LIN {X 0,Y 574.65,Z 406.368,A -85,B 0,C 180,E1 -1993.417,E2 -1993.417} C_VEL
LIN {X 0,Y 574.045,Z 400.558,A -85,B 0,C 180,E1 -1993.505,E2 -1993.505} C_VEL
LIN {X 0,Y 573.916,Z 376.535,A -85,B 0,C 180,E1 -1993.811,E2 -1993.811} C_VEL
LIN {X 0,Y 573.362,Z 372.933,A -85,B 0,C 180,E1 -1993.874,E2 -1993.874} C_VEL
LIN {X 0,Y 573.52,Z 353.065,A -85,B 0,C 180,E1 -1996.97,E2 -1996.97} C_VEL
LIN {X 0,Y 573.745,Z 333.535,A -85,B 0,C 180,E1 -2000.059,E2 -2000.059} C_VEL
LIN {X 0,Y 573.574,Z 324.195,A -85,B 0,C 180,E1 -2001.567,E2 -2001.567} C_VEL
LIN {X 0,Y 573.285,Z 322.702,A -85,B 0,C 180,E1 -2001.838,E2 -2001.838} C_VEL
LIN {X 0,Y 573.272,Z 322.698,A -85,B 0,C 180,E1 -2004.878,E2 -2004.878} C_VEL
LIN {X 0,Y 573.27,Z 322.699,A -85,B 0,C 180,E1 -2007.766,E2 -2007.766} C_VEL
LIN {X 0,Y 573.249,Z 322.707,A -85,B 0,C 180,E1 -2010.176,E2 -2010.176} C_VEL
LIN {X 0,Y 573.257,Z 322.699,A -85,B 0,C 180,E1 -2012.645,E2 -2012.645} C_VEL
LIN {X 0,Y 573.209,Z 322.704,A -85,B 0,C 180,E1 -2015.188,E2 -2015.188} C_VEL
LIN {X 0,Y 573.234,Z 322.708,A -85,B 0,C 180,E1 -2017.808,E2 -2017.808} C_VEL
LIN {X 0,Y 573.25,Z 322.699,A -85,B 0,C 180,E1 -2020.525,E2 -2020.525} C_VEL
LIN {X 0,Y 573.24,Z 322.708,A -85,B 0,C 180,E1 -2023.668,E2 -2023.668} C_VEL
LIN {X 0,Y 573.212,Z 322.703,A -85,B 0,C 180,E1 -2026.638,E2 -2026.638} C_VEL
LIN {X 0,Y 573.25,Z 322.706,A -85,B 0,C 180,E1 -2029.475,E2 -2029.475} C_VEL
LIN {X 0,Y 573.22,Z 322.703,A -85,B 0,C 180,E1 -2032.19,E2 -2032.19} C_VEL
LIN {X 0,Y 573.227,Z 322.708,A -85,B 0,C 180,E1 -2035.23,E2 -2035.23} C_VEL
LIN {X 0,Y 573.223,Z 322.703,A -85,B 0,C 180,E1 -2038.183,E2 -2038.183} C_VEL
LIN {X 0,Y 573.229,Z 322.703,A -85,B 0,C 180,E1 -2040.631,E2 -2040.631} C_VEL
LIN {X 0,Y 573.188,Z 322.712,A -85,B 0,C 180,E1 -2043.518,E2 -2043.518} C_VEL
LIN {X 0,Y 573.189,Z 322.708,A -85,B 0,C 180,E1 -2046.132,E2 -2046.132} C_VEL
LIN {X 0,Y 573.225,Z 322.734,A -85,B 0,C 180,E1 -2047.471,E2 -2047.471} C_VEL
LIN {X 0,Y 573.941,Z 327.822,A -85,B 0,C 180,E1 -2048.258,E2 -2048.258} C_VEL
LIN {X 0,Y 573.725,Z 345.632,A -85,B 0,C 180,E1 -2050.871,E2 -2050.871} C_VEL
LIN {X 0,Y 573.558,Z 362.355,A -85,B 0,C 180,E1 -2053.29,E2 -2053.29} C_VEL
LIN {X 0,Y 574.612,Z 367.973,A -85,B 0,C 180,E1 -2053.394,E2 -2053.394} C_VEL
LIN {X 0,Y 574.27,Z 498.274,A -85,B 0,C 180,E1 -2055.062,E2 -2055.062} C_VEL
LIN {X 0,Y 574.177,Z 511.252,A -85,B 0,C 180,E1 -2055.339,E2 -2055.339} C_VEL
LIN {X 0,Y 574.09,Z 525.101,A -85,B 0,C 180,E1 -2055.771,E2 -2055.771} C_VEL
LIN {X 0,Y 573.918,Z 538.916,A -85,B 0,C 180,E1 -2056.365,E2 -2056.365} C_VEL
LIN {X 0,Y 573.741,Z 550.437,A -85,B 0,C 180,E1 -2056.991,E2 -2056.991} C_VEL
LIN {X 0,Y 573.601,Z 561.254,A -85,B 0,C 180,E1 -2057.708,E2 -2057.708} C_VEL
LIN {X 0,Y 573.455,Z 571.619,A -85,B 0,C 180,E1 -2058.53,E2 -2058.53} C_VEL
LIN {X 0,Y 573.355,Z 580.918,A -85,B 0,C 180,E1 -2059.404,E2 -2059.404} C_VEL
LIN {X 0,Y 573.256,Z 590.452,A -85,B 0,C 180,E1 -2060.472,E2 -2060.472} C_VEL
LIN {X 0,Y 573.143,Z 599.468,A -85,B 0,C 180,E1 -2061.715,E2 -2061.715} C_VEL
LIN {X 0,Y 573.091,Z 604.887,A -85,B 0,C 180,E1 -2062.601,E2 -2062.601} C_VEL
LIN {X 0,Y 573.022,Z 610.311,A -85,B 0,C 180,E1 -2063.662,E2 -2063.662} C_VEL
LIN {X 0,Y 573,Z 614.764,A -85,B 0,C 180,E1 -2064.721,E2 -2064.721} C_VEL
LIN {X 0,Y 573.029,Z 618.315,A -85,B 0,C 180,E1 -2065.779,E2 -2065.779} C_VEL
LIN {X 0,Y 572.957,Z 621.715,A -85,B 0,C 180,E1 -2067.187,E2 -2067.187} C_VEL
LIN {X 0,Y 572.939,Z 622.942,A -85,B 0,C 180,E1 -2067.89,E2 -2067.89} C_VEL
LIN {X 0,Y 572.936,Z 624.281,A -85,B 0,C 180,E1 -2069.296,E2 -2069.296} C_VEL
LIN {X 0,Y 572.937,Z 624.496,A -85,B 0,C 180,E1 -2069.999,E2 -2069.999} C_VEL
LIN {X 0,Y 572.941,Z 623.863,A -85,B 0,C 180,E1 -2071.405,E2 -2071.405} C_VEL
LIN {X 0,Y 572.954,Z 621.893,A -85,B 0,C 180,E1 -2072.811,E2 -2072.811} C_VEL
LIN {X 0,Y 573.008,Z 620.437,A -85,B 0,C 180,E1 -2073.515,E2 -2073.515} C_VEL
LIN {X 0,Y 572.955,Z 616.342,A -85,B 0,C 180,E1 -2074.925,E2 -2074.925} C_VEL
LIN {X 0,Y 573.044,Z 612.299,A -85,B 0,C 180,E1 -2075.983,E2 -2075.983} C_VEL
LIN {X 0,Y 573.052,Z 607.286,A -85,B 0,C 180,E1 -2077.043,E2 -2077.043} C_VEL
LIN {X 0,Y 573.128,Z 601.186,A -85,B 0,C 180,E1 -2078.106,E2 -2078.106} C_VEL
LIN {X 0,Y 573.219,Z 593.877,A -85,B 0,C 180,E1 -2079.17,E2 -2079.17} C_VEL
LIN {X 0,Y 573.303,Z 585.125,A -85,B 0,C 180,E1 -2080.238,E2 -2080.238} C_VEL
LIN {X 0,Y 573.486,Z 573.884,A -85,B 0,C 180,E1 -2081.365,E2 -2081.365} C_VEL
LIN {X 0,Y 573.584,Z 562.523,A -85,B 0,C 180,E1 -2082.291,E2 -2082.291} C_VEL
LIN {X 0,Y 573.731,Z 551.933,A -85,B 0,C 180,E1 -2083.007,E2 -2083.007} C_VEL
LIN {X 0,Y 573.879,Z 540.703,A -85,B 0,C 180,E1 -2083.634,E2 -2083.634} C_VEL
LIN {X 0,Y 574.011,Z 528.847,A -85,B 0,C 180,E1 -2084.173,E2 -2084.173} C_VEL
LIN {X 0,Y 574.173,Z 513.454,A -85,B 0,C 180,E1 -2084.696,E2 -2084.696} C_VEL
LIN {X 0,Y 574.271,Z 499.72,A -85,B 0,C 180,E1 -2085.004,E2 -2085.004} C_VEL
LIN {X 0,Y 574.432,Z 453.324,A -85,B 0,C 180,E1 -2085.613,E2 -2085.613} C_VEL
LIN {X 0,Y 574.556,Z 367.642,A -85,B 0,C 180,E1 -2086.702,E2 -2086.702} C_VEL
LIN {X 0,Y 573.565,Z 362.258,A -85,B 0,C 180,E1 -2086.813,E2 -2086.813} C_VEL
LIN {X 0,Y 573.811,Z 341.174,A -85,B 0,C 180,E1 -2089.868,E2 -2089.868} C_VEL
LIN {X 0,Y 573.911,Z 327.171,A -85,B 0,C 180,E1 -2091.93,E2 -2091.93} C_VEL
LIN {X 0,Y 573.224,Z 322.71,A -85,B 0,C 180,E1 -2092.646,E2 -2092.646} C_VEL
LIN {X 0,Y 573.215,Z 322.707,A -85,B 0,C 180,E1 -2095.41,E2 -2095.41} C_VEL
LIN {X 0,Y 573.193,Z 322.71,A -85,B 0,C 180,E1 -2098.565,E2 -2098.565} C_VEL
LIN {X 0,Y 573.205,Z 322.714,A -85,B 0,C 180,E1 -2100.993,E2 -2100.993} C_VEL
LIN {X 0,Y 573.235,Z 322.703,A -85,B 0,C 180,E1 -2103.519,E2 -2103.519} C_VEL
LIN {X 0,Y 573.184,Z 322.707,A -85,B 0,C 180,E1 -2106.052,E2 -2106.052} C_VEL
LIN {X 0,Y 573.222,Z 322.708,A -85,B 0,C 180,E1 -2108.701,E2 -2108.701} C_VEL
LIN {X 0,Y 573.192,Z 322.707,A -85,B 0,C 180,E1 -2111.458,E2 -2111.458} C_VEL
LIN {X 0,Y 573.206,Z 322.705,A -85,B 0,C 180,E1 -2114.334,E2 -2114.334} C_VEL
LIN {X 0,Y 573.218,Z 322.708,A -85,B 0,C 180,E1 -2116.639,E2 -2116.639} C_VEL
LIN {X 0,Y 573.234,Z 322.701,A -85,B 0,C 180,E1 -2119.474,E2 -2119.474} C_VEL
LIN {X 0,Y 573.209,Z 322.703,A -85,B 0,C 180,E1 -2122.19,E2 -2122.19} C_VEL
LIN {X 0,Y 573.208,Z 322.706,A -85,B 0,C 180,E1 -2125.23,E2 -2125.23} C_VEL
LIN {X 0,Y 573.223,Z 322.699,A -85,B 0,C 180,E1 -2127.773,E2 -2127.773} C_VEL
LIN {X 0,Y 573.218,Z 322.71,A -85,B 0,C 180,E1 -2130.631,E2 -2130.631} C_VEL
LIN {X 0,Y 573.194,Z 322.702,A -85,B 0,C 180,E1 -2133.513,E2 -2133.513} C_VEL
LIN {X 0,Y 573.181,Z 322.708,A -85,B 0,C 180,E1 -2136.132,E2 -2136.132} C_VEL
LIN {X 0,Y 573.236,Z 322.708,A -85,B 0,C 180,E1 -2138.709,E2 -2138.709} C_VEL
LIN {X 0,Y 573.183,Z 322.705,A -85,B 0,C 180,E1 -2141.41,E2 -2141.41} C_VEL
LIN {X 0,Y 573.206,Z 322.703,A -85,B 0,C 180,E1 -2143.62,E2 -2143.62} C_VEL
LIN {X 0,Y 573.182,Z 322.714,A -85,B 0,C 180,E1 -2146.528,E2 -2146.528} C_VEL
LIN {X 0,Y 573.22,Z 322.702,A -85,B 0,C 180,E1 -2149.402,E2 -2149.402} C_VEL
LIN {X 0,Y 573.244,Z 322.702,A -85,B 0,C 180,E1 -2152.249,E2 -2152.249} C_VEL
LIN {X 0,Y 573.266,Z 322.698,A -85,B 0,C 180,E1 -2155.077,E2 -2155.077} C_VEL
LIN {X 0,Y 573.27,Z 322.696,A -85,B 0,C 180,E1 -2157.892,E2 -2157.892} C_VEL
LIN {X 0,Y 573.316,Z 322.697,A -85,B 0,C 180,E1 -2160.702,E2 -2160.702} C_VEL
LIN {X 0,Y 573.282,Z 322.699,A -85,B 0,C 180,E1 -2162.811,E2 -2162.811} C_VEL
LIN {X 0,Y 573.243,Z 322.698,A -85,B 0,C 180,E1 -2165.629,E2 -2165.629} C_VEL
LIN {X 0,Y 573.22,Z 322.711,A -85,B 0,C 180,E1 -2168.46,E2 -2168.46} C_VEL
LIN {X 0,Y 573.219,Z 322.702,A -85,B 0,C 180,E1 -2171.313,E2 -2171.313} C_VEL
LIN {X 0,Y 573.261,Z 322.706,A -85,B 0,C 180,E1 -2174.423,E2 -2174.423} C_VEL
LIN {X 0,Y 573.202,Z 322.704,A -85,B 0,C 180,E1 -2177.113,E2 -2177.113} C_VEL
LIN {X 0,Y 573.219,Z 322.706,A -85,B 0,C 180,E1 -2180.078,E2 -2180.078} C_VEL
LIN {X 0,Y 573.21,Z 322.71,A -85,B 0,C 180,E1 -2182.339,E2 -2182.339} C_VEL
LIN {X 0,Y 573.193,Z 322.708,A -85,B 0,C 180,E1 -2184.866,E2 -2184.866} C_VEL
LIN {X 0,Y 573.216,Z 322.703,A -85,B 0,C 180,E1 -2187.769,E2 -2187.769} C_VEL
LIN {X 0,Y 573.209,Z 322.708,A -85,B 0,C 180,E1 -2190.178,E2 -2190.178} C_VEL
LIN {X 0,Y 573.231,Z 322.705,A -85,B 0,C 180,E1 -2192.647,E2 -2192.647} C_VEL
LIN {X 0,Y 573.169,Z 322.708,A -85,B 0,C 180,E1 -2195.191,E2 -2195.191} C_VEL
LIN {X 0,Y 573.202,Z 322.707,A -85,B 0,C 180,E1 -2197.81,E2 -2197.81} C_VEL
LIN {X 0,Y 573.188,Z 322.711,A -85,B 0,C 180,E1 -2200.53,E2 -2200.53} C_VEL
LIN {X 0,Y 573.186,Z 322.706,A -85,B 0,C 180,E1 -2203.364,E2 -2203.364} C_VEL
LIN {X 0,Y 573.182,Z 322.715,A -85,B 0,C 180,E1 -2206.338,E2 -2206.338} C_VEL
LIN {X 0,Y 573.178,Z 322.712,A -85,B 0,C 180,E1 -2208.54,E2 -2208.54} C_VEL
LIN {X 0,Y 573.204,Z 322.704,A -85,B 0,C 180,E1 -2211.297,E2 -2211.297} C_VEL
LIN {X 0,Y 573.173,Z 322.715,A -85,B 0,C 180,E1 -2214.024,E2 -2214.024} C_VEL
LIN {X 0,Y 573.213,Z 322.708,A -85,B 0,C 180,E1 -2216.516,E2 -2216.516} C_VEL
LIN {X 0,Y 573.209,Z 322.703,A -85,B 0,C 180,E1 -2219.121,E2 -2219.121} C_VEL
LIN {X 0,Y 573.184,Z 322.714,A -85,B 0,C 180,E1 -2221.984,E2 -2221.984} C_VEL
LIN {X 0,Y 573.199,Z 322.71,A -85,B 0,C 180,E1 -2224.589,E2 -2224.589} C_VEL
LIN {X 0,Y 573.241,Z 322.841,A -85,B 0,C 180,E1 -2226.382,E2 -2226.382} C_VEL
LIN {X 0,Y 574.048,Z 327.852,A -85,B 0,C 180,E1 -2227.127,E2 -2227.127} C_VEL
LIN {X 0,Y 573.904,Z 345.308,A -85,B 0,C 180,E1 -2229.575,E2 -2229.575} C_VEL
LIN {X 0,Y 573.681,Z 367.06,A -85,B 0,C 180,E1 -2232.572,E2 -2232.572} C_VEL
LIN {X 0,Y 573.602,Z 371.957,A -85,B 0,C 180,E1 -2233.239,E2 -2233.239} C_VEL
LIN {X 0,Y 574.57,Z 377.542,A -85,B 0,C 180,E1 -2233.342,E2 -2233.342} C_VEL
LIN {X 0,Y 574.302,Z 508.713,A -85,B 0,C 180,E1 -2235.019,E2 -2235.019} C_VEL
LIN {X 0,Y 574.171,Z 523.157,A -85,B 0,C 180,E1 -2235.341,E2 -2235.341} C_VEL
LIN {X 0,Y 574.023,Z 537.735,A -85,B 0,C 180,E1 -2235.827,E2 -2235.827} C_VEL
LIN {X 0,Y 573.874,Z 551.669,A -85,B 0,C 180,E1 -2236.456,E2 -2236.456} C_VEL
LIN {X 0,Y 573.718,Z 564.121,A -85,B 0,C 180,E1 -2237.173,E2 -2237.173} C_VEL
LIN {X 0,Y 573.532,Z 576.658,A -85,B 0,C 180,E1 -2238.067,E2 -2238.067} C_VEL
LIN {X 0,Y 573.435,Z 588.188,A -85,B 0,C 180,E1 -2239.085,E2 -2239.085} C_VEL
LIN {X 0,Y 573.239,Z 597.861,A -85,B 0,C 180,E1 -2240.118,E2 -2240.118} C_VEL
LIN {X 0,Y 573.201,Z 606.18,A -85,B 0,C 180,E1 -2241.185,E2 -2241.185} C_VEL
LIN {X 0,Y 573.109,Z 614.134,A -85,B 0,C 180,E1 -2242.426,E2 -2242.426} C_VEL
LIN {X 0,Y 573.02,Z 620.532,A -85,B 0,C 180,E1 -2243.664,E2 -2243.664} C_VEL
LIN {X 0,Y 573.001,Z 624.964,A -85,B 0,C 180,E1 -2244.723,E2 -2244.723} C_VEL
LIN {X 0,Y 573.028,Z 628.448,A -85,B 0,C 180,E1 -2245.781,E2 -2245.781} C_VEL
LIN {X 0,Y 572.956,Z 631.836,A -85,B 0,C 180,E1 -2247.189,E2 -2247.189} C_VEL
LIN {X 0,Y 572.941,Z 633.834,A -85,B 0,C 180,E1 -2248.595,E2 -2248.595} C_VEL
LIN {X 0,Y 572.937,Z 634.5,A -85,B 0,C 180,E1 -2250.001,E2 -2250.001} C_VEL
LIN {X 0,Y 572.941,Z 633.831,A -85,B 0,C 180,E1 -2251.407,E2 -2251.407} C_VEL
LIN {X 0,Y 572.956,Z 631.83,A -85,B 0,C 180,E1 -2252.813,E2 -2252.813} C_VEL
LIN {X 0,Y 573.028,Z 628.44,A -85,B 0,C 180,E1 -2254.221,E2 -2254.221} C_VEL
LIN {X 0,Y 573.055,Z 623.565,A -85,B 0,C 180,E1 -2255.631,E2 -2255.631} C_VEL
LIN {X 0,Y 573.059,Z 618.849,A -85,B 0,C 180,E1 -2256.694,E2 -2256.694} C_VEL
LIN {X 0,Y 573.126,Z 612.031,A -85,B 0,C 180,E1 -2257.93,E2 -2257.93} C_VEL
LIN {X 0,Y 573.226,Z 603.551,A -85,B 0,C 180,E1 -2259.172,E2 -2259.172} C_VEL
LIN {X 0,Y 573.305,Z 594.698,A -85,B 0,C 180,E1 -2260.24,E2 -2260.24} C_VEL
LIN {X 0,Y 573.464,Z 583.98,A -85,B 0,C 180,E1 -2261.309,E2 -2261.309} C_VEL
LIN {X 0,Y 573.618,Z 573.129,A -85,B 0,C 180,E1 -2262.202,E2 -2262.202} C_VEL
LIN {X 0,Y 573.74,Z 561.241,A -85,B 0,C 180,E1 -2263.009,E2 -2263.009} C_VEL
LIN {X 0,Y 573.957,Z 548.078,A -85,B 0,C 180,E1 -2263.725,E2 -2263.725} C_VEL
LIN {X 0,Y 574.104,Z 534.807,A -85,B 0,C 180,E1 -2264.285,E2 -2264.285} C_VEL
LIN {X 0,Y 574.204,Z 520.768,A -85,B 0,C 180,E1 -2264.721,E2 -2264.721} C_VEL
LIN {X 0,Y 574.309,Z 507.071,A -85,B 0,C 180,E1 -2265.005,E2 -2265.005} C_VEL
LIN {X 0,Y 574.472,Z 376.673,A -85,B 0,C 180,E1 -2266.672,E2 -2266.672} C_VEL
LIN {X 0,Y 573.592,Z 371.839,A -85,B 0,C 180,E1 -2266.777,E2 -2266.777} C_VEL
LIN {X 0,Y 573.841,Z 350.931,A -85,B 0,C 180,E1 -2269.646,E2 -2269.646} C_VEL
LIN {X 0,Y 574.092,Z 330.521,A -85,B 0,C 180,E1 -2272.493,E2 -2272.493} C_VEL
LIN {X 0,Y 573.715,Z 325.251,A -85,B 0,C 180,E1 -2273.256,E2 -2273.256} C_VEL
LIN {X 0,Y 573.228,Z 322.711,A -85,B 0,C 180,E1 -2273.643,E2 -2273.643} C_VEL
LIN {X 0,Y 573.201,Z 322.707,A -85,B 0,C 180,E1 -2276.485,E2 -2276.485} C_VEL
LIN {X 0,Y 573.225,Z 322.709,A -85,B 0,C 180,E1 -2279.369,E2 -2279.369} C_VEL
LIN {X 0,Y 573.241,Z 322.701,A -85,B 0,C 180,E1 -2282.226,E2 -2282.226} C_VEL
LIN {X 0,Y 573.234,Z 322.703,A -85,B 0,C 180,E1 -2284.771,E2 -2284.771} C_VEL
LIN {X 0,Y 573.234,Z 322.702,A -85,B 0,C 180,E1 -2287.808,E2 -2287.808} C_VEL
LIN {X 0,Y 573.249,Z 322.701,A -85,B 0,C 180,E1 -2290.526,E2 -2290.526} C_VEL
LIN {X 0,Y 573.241,Z 322.703,A -85,B 0,C 180,E1 -2293.36,E2 -2293.36} C_VEL
LIN {X 0,Y 573.249,Z 322.702,A -85,B 0,C 180,E1 -2296.331,E2 -2296.331} C_VEL
LIN {X 0,Y 573.234,Z 322.708,A -85,B 0,C 180,E1 -2298.543,E2 -2298.543} C_VEL
LIN {X 0,Y 573.242,Z 322.7,A -85,B 0,C 180,E1 -2301.298,E2 -2301.298} C_VEL
LIN {X 0,Y 573.198,Z 322.709,A -85,B 0,C 180,E1 -2304.021,E2 -2304.021} C_VEL
LIN {X 0,Y 573.274,Z 322.702,A -85,B 0,C 180,E1 -2306.518,E2 -2306.518} C_VEL
LIN {X 0,Y 573.23,Z 322.702,A -85,B 0,C 180,E1 -2309.119,E2 -2309.119} C_VEL
LIN {X 0,Y 573.227,Z 322.705,A -85,B 0,C 180,E1 -2311.435,E2 -2311.435} C_VEL
LIN {X 0,Y 573.225,Z 322.704,A -85,B 0,C 180,E1 -2314.589,E2 -2314.589} C_VEL
LIN {X 0,Y 573.221,Z 322.712,A -85,B 0,C 180,E1 -2317.662,E2 -2317.662} C_VEL
LIN {X 0,Y 573.233,Z 322.723,A -85,B 0,C 180,E1 -2318.278,E2 -2318.278} C_VEL
LIN {X 0,Y 573.78,Z 328.306,A -85,B 0,C 180,E1 -2319.194,E2 -2319.194} C_VEL
LIN {X 0,Y 573.558,Z 346.975,A -85,B 0,C 180,E1 -2322.162,E2 -2322.162} C_VEL
LIN {X 0,Y 573.397,Z 365.644,A -85,B 0,C 180,E1 -2325.085,E2 -2325.085} C_VEL
LIN {X 0,Y 573.36,Z 372.937,A -85,B 0,C 180,E1 -2326.216,E2 -2326.216} C_VEL
LIN {X 0,Y 574.089,Z 378.02,A -85,B 0,C 180,E1 -2326.302,E2 -2326.302} C_VEL
LIN {X 0,Y 573.881,Z 480.361,A -85,B 0,C 180,E1 -2327.602,E2 -2327.602} C_VEL
LIN {X 0,Y 573.814,Z 493.729,A -85,B 0,C 180,E1 -2327.915,E2 -2327.915} C_VEL
LIN {X 0,Y 573.704,Z 505.856,A -85,B 0,C 180,E1 -2328.339,E2 -2328.339} C_VEL
LIN {X 0,Y 573.62,Z 517.359,A -85,B 0,C 180,E1 -2328.878,E2 -2328.878} C_VEL
LIN {X 0,Y 573.437,Z 529.062,A -85,B 0,C 180,E1 -2329.585,E2 -2329.585} C_VEL
LIN {X 0,Y 573.329,Z 539.551,A -85,B 0,C 180,E1 -2330.386,E2 -2330.386} C_VEL
LIN {X 0,Y 573.243,Z 548.164,A -85,B 0,C 180,E1 -2331.185,E2 -2331.185} C_VEL
LIN {X 0,Y 573.162,Z 556.072,A -85,B 0,C 180,E1 -2332.071,E2 -2332.071} C_VEL
LIN {X 0,Y 573.089,Z 564.072,A -85,B 0,C 180,E1 -2333.169,E2 -2333.169} C_VEL
LIN {X 0,Y 573.071,Z 570.943,A -85,B 0,C 180,E1 -2334.37,E2 -2334.37} C_VEL
LIN {X 0,Y 573.028,Z 575.704,A -85,B 0,C 180,E1 -2335.428,E2 -2335.428} C_VEL
LIN {X 0,Y 573.023,Z 579.31,A -85,B 0,C 180,E1 -2336.484,E2 -2336.484} C_VEL
LIN {X 0,Y 572.959,Z 581.18,A -85,B 0,C 180,E1 -2337.188,E2 -2337.188} C_VEL
LIN {X 0,Y 572.938,Z 582.612,A -85,B 0,C 180,E1 -2337.891,E2 -2337.891} C_VEL
LIN {X 0,Y 572.947,Z 583.637,A -85,B 0,C 180,E1 -2338.594,E2 -2338.594} C_VEL
LIN {X 0,Y 572.941,Z 584.265,A -85,B 0,C 180,E1 -2339.297,E2 -2339.297} C_VEL
LIN {X 0,Y 572.938,Z 584.496,A -85,B 0,C 180,E1 -2340,E2 -2340} C_VEL
LIN {X 0,Y 572.941,Z 584.321,A -85,B 0,C 180,E1 -2340.703,E2 -2340.703} C_VEL
LIN {X 0,Y 572.946,Z 583.737,A -85,B 0,C 180,E1 -2341.406,E2 -2341.406} C_VEL
LIN {X 0,Y 572.96,Z 581.385,A -85,B 0,C 180,E1 -2342.812,E2 -2342.812} C_VEL
LIN {X 0,Y 573.015,Z 578.525,A -85,B 0,C 180,E1 -2343.868,E2 -2343.868} C_VEL
LIN {X 0,Y 572.963,Z 574.637,A -85,B 0,C 180,E1 -2344.926,E2 -2344.926} C_VEL
LIN {X 0,Y 573.073,Z 569.578,A -85,B 0,C 180,E1 -2345.984,E2 -2345.984} C_VEL
LIN {X 0,Y 573.084,Z 563.263,A -85,B 0,C 180,E1 -2347.044,E2 -2347.044} C_VEL
LIN {X 0,Y 573.175,Z 555.37,A -85,B 0,C 180,E1 -2348.106,E2 -2348.106} C_VEL
LIN {X 0,Y 573.251,Z 547.284,A -85,B 0,C 180,E1 -2348.993,E2 -2348.993} C_VEL
LIN {X 0,Y 573.337,Z 537.447,A -85,B 0,C 180,E1 -2349.882,E2 -2349.882} C_VEL
LIN {X 0,Y 573.488,Z 526.382,A -85,B 0,C 180,E1 -2350.681,E2 -2350.681} C_VEL
LIN {X 0,Y 573.615,Z 514.134,A -85,B 0,C 180,E1 -2351.378,E2 -2351.378} C_VEL
LIN {X 0,Y 573.729,Z 501.526,A -85,B 0,C 180,E1 -2351.921,E2 -2351.921} C_VEL
LIN {X 0,Y 573.841,Z 488.808,A -85,B 0,C 180,E1 -2352.309,E2 -2352.309} C_VEL
LIN {X 0,Y 573.924,Z 476.185,A -85,B 0,C 180,E1 -2352.554,E2 -2352.554} C_VEL
LIN {X 0,Y 574.045,Z 400.558,A -85,B 0,C 180,E1 -2353.505,E2 -2353.505} C_VEL
LIN {X 0,Y 573.415,Z 396.677,A -85,B 0,C 180,E1 -2353.569,E2 -2353.569} C_VEL
LIN {X 0,Y 567.854,Z 384.698,A -85,B 0,C 180,E1 -2353.857,E2 -2353.857} C_VEL
LIN {X 0,Y 567.217,Z 380.817,A -85,B 0,C 180,E1 -2353.922,E2 -2353.922} C_VEL
LIN {X 0,Y 566.613,Z 374.676,A -85,B 0,C 180,E1 -2354.016,E2 -2354.016} C_VEL
LIN {X 0,Y 566.336,Z 372.93,A -85,B 0,C 180,E1 -2354.05,E2 -2354.05} C_VEL
LIN {X 0,Y 566.527,Z 354.911,A -85,B 0,C 180,E1 -2356.891,E2 -2356.891} C_VEL
LIN {X 0,Y 566.743,Z 335.855,A -85,B 0,C 180,E1 -2359.939,E2 -2359.939} C_VEL
LIN {X 0,Y 566.66,Z 325.953,A -85,B 0,C 180,E1 -2361.535,E2 -2361.535} C_VEL
LIN {X 0,Y 566.222,Z 323.582,A -85,B 0,C 180,E1 -2361.957,E2 -2361.957} C_VEL
LIN {X 0,Y 566.224,Z 323.575,A -85,B 0,C 180,E1 -2365.03,E2 -2365.03} C_VEL
LIN {X 0,Y 566.198,Z 323.577,A -85,B 0,C 180,E1 -2367.34,E2 -2367.34} C_VEL
LIN {X 0,Y 566.205,Z 323.58,A -85,B 0,C 180,E1 -2369.769,E2 -2369.769} C_VEL
LIN {X 0,Y 566.206,Z 323.58,A -85,B 0,C 180,E1 -2372.429,E2 -2372.429} C_VEL
LIN {X 0,Y 566.182,Z 323.579,A -85,B 0,C 180,E1 -2374.989,E2 -2374.989} C_VEL
LIN {X 0,Y 566.196,Z 323.58,A -85,B 0,C 180,E1 -2377.461,E2 -2377.461} C_VEL
LIN {X 0,Y 566.212,Z 323.579,A -85,B 0,C 180,E1 -2380.199,E2 -2380.199} C_VEL
LIN {X 0,Y 566.197,Z 323.578,A -85,B 0,C 180,E1 -2383.055,E2 -2383.055} C_VEL
LIN {X 0,Y 566.163,Z 323.585,A -85,B 0,C 180,E1 -2386.053,E2 -2386.053} C_VEL
LIN {X 0,Y 566.161,Z 323.582,A -85,B 0,C 180,E1 -2388.858,E2 -2388.858} C_VEL
LIN {X 0,Y 566.204,Z 323.584,A -85,B 0,C 180,E1 -2391.443,E2 -2391.443} C_VEL
LIN {X 0,Y 566.146,Z 323.584,A -85,B 0,C 180,E1 -2394.306,E2 -2394.306} C_VEL
LIN {X 0,Y 566.166,Z 323.584,A -85,B 0,C 180,E1 -2396.893,E2 -2396.893} C_VEL
LIN {X 0,Y 566.162,Z 323.59,A -85,B 0,C 180,E1 -2399.405,E2 -2399.405} C_VEL
LIN {X 0,Y 566.153,Z 323.585,A -85,B 0,C 180,E1 -2401.853,E2 -2401.853} C_VEL
LIN {X 0,Y 566.163,Z 323.583,A -85,B 0,C 180,E1 -2404.248,E2 -2404.248} C_VEL
LIN {X 0,Y 566.229,Z 323.751,A -85,B 0,C 180,E1 -2407.324,E2 -2407.324} C_VEL
LIN {X 0,Y 567.036,Z 329.112,A -85,B 0,C 180,E1 -2408.171,E2 -2408.171} C_VEL
LIN {X 0,Y 566.777,Z 346.967,A -85,B 0,C 180,E1 -2410.824,E2 -2410.824} C_VEL
LIN {X 0,Y 566.592,Z 362.372,A -85,B 0,C 180,E1 -2413.079,E2 -2413.079} C_VEL
LIN {X 0,Y 567.808,Z 369.08,A -85,B 0,C 180,E1 -2413.203,E2 -2413.203} C_VEL
LIN {X 0,Y 567.41,Z 498.252,A -85,B 0,C 180,E1 -2414.877,E2 -2414.877} C_VEL
LIN {X 0,Y 567.293,Z 510.708,A -85,B 0,C 180,E1 -2415.143,E2 -2415.143} C_VEL
LIN {X 0,Y 567.213,Z 523.724,A -85,B 0,C 180,E1 -2415.545,E2 -2415.545} C_VEL
LIN {X 0,Y 567.062,Z 537.144,A -85,B 0,C 180,E1 -2416.105,E2 -2416.105} C_VEL
LIN {X 0,Y 566.813,Z 548.969,A -85,B 0,C 180,E1 -2416.738,E2 -2416.738} C_VEL
LIN {X 0,Y 566.65,Z 560.011,A -85,B 0,C 180,E1 -2417.463,E2 -2417.463} C_VEL
LIN {X 0,Y 566.503,Z 570.347,A -85,B 0,C 180,E1 -2418.278,E2 -2418.278} C_VEL
LIN {X 0,Y 566.4,Z 579.453,A -85,B 0,C 180,E1 -2419.125,E2 -2419.125} C_VEL
LIN {X 0,Y 566.199,Z 588.971,A -85,B 0,C 180,E1 -2420.172,E2 -2420.172} C_VEL
LIN {X 0,Y 566.091,Z 598.332,A -85,B 0,C 180,E1 -2421.431,E2 -2421.431} C_VEL
LIN {X 0,Y 566.017,Z 604.886,A -85,B 0,C 180,E1 -2422.508,E2 -2422.508} C_VEL
LIN {X 0,Y 565.946,Z 610.312,A -85,B 0,C 180,E1 -2423.582,E2 -2423.582} C_VEL
LIN {X 0,Y 565.928,Z 614.759,A -85,B 0,C 180,E1 -2424.655,E2 -2424.655} C_VEL
LIN {X 0,Y 565.957,Z 618.316,A -85,B 0,C 180,E1 -2425.726,E2 -2425.726} C_VEL
LIN {X 0,Y 565.875,Z 621.709,A -85,B 0,C 180,E1 -2427.151,E2 -2427.151} C_VEL
LIN {X 0,Y 565.84,Z 622.944,A -85,B 0,C 180,E1 -2427.864,E2 -2427.864} C_VEL
LIN {X 0,Y 565.836,Z 624.273,A -85,B 0,C 180,E1 -2429.287,E2 -2429.287} C_VEL
LIN {X 0,Y 565.838,Z 624.496,A -85,B 0,C 180,E1 -2429.999,E2 -2429.999} C_VEL
LIN {X 0,Y 565.841,Z 623.859,A -85,B 0,C 180,E1 -2431.422,E2 -2431.422} C_VEL
LIN {X 0,Y 565.873,Z 621.884,A -85,B 0,C 180,E1 -2432.846,E2 -2432.846} C_VEL
LIN {X 0,Y 565.914,Z 620.437,A -85,B 0,C 180,E1 -2433.559,E2 -2433.559} C_VEL
LIN {X 0,Y 565.929,Z 617.534,A -85,B 0,C 180,E1 -2434.629,E2 -2434.629} C_VEL
LIN {X 0,Y 565.961,Z 612.288,A -85,B 0,C 180,E1 -2436.058,E2 -2436.058} C_VEL
LIN {X 0,Y 565.979,Z 607.274,A -85,B 0,C 180,E1 -2437.132,E2 -2437.132} C_VEL
LIN {X 0,Y 566.055,Z 601.175,A -85,B 0,C 180,E1 -2438.208,E2 -2438.208} C_VEL
LIN {X 0,Y 566.171,Z 593.863,A -85,B 0,C 180,E1 -2439.285,E2 -2439.285} C_VEL
LIN {X 0,Y 566.282,Z 585.109,A -85,B 0,C 180,E1 -2440.366,E2 -2440.366} C_VEL
LIN {X 0,Y 566.467,Z 573.529,A -85,B 0,C 180,E1 -2441.539,E2 -2441.539} C_VEL
LIN {X 0,Y 566.623,Z 562.501,A -85,B 0,C 180,E1 -2442.444,E2 -2442.444} C_VEL
LIN {X 0,Y 566.762,Z 551.907,A -85,B 0,C 180,E1 -2443.17,E2 -2443.17} C_VEL
LIN {X 0,Y 566.951,Z 540.679,A -85,B 0,C 180,E1 -2443.804,E2 -2443.804} C_VEL
LIN {X 0,Y 567.125,Z 528.81,A -85,B 0,C 180,E1 -2444.349,E2 -2444.349} C_VEL
LIN {X 0,Y 567.303,Z 513.953,A -85,B 0,C 180,E1 -2444.864,E2 -2444.864} C_VEL
LIN {X 0,Y 567.422,Z 499.629,A -85,B 0,C 180,E1 -2445.19,E2 -2445.19} C_VEL
LIN {X 0,Y 567.573,Z 456.856,A -85,B 0,C 180,E1 -2445.761,E2 -2445.761} C_VEL
LIN {X 0,Y 567.719,Z 368.414,A -85,B 0,C 180,E1 -2446.898,E2 -2446.898} C_VEL
LIN {X 0,Y 566.585,Z 362.233,A -85,B 0,C 180,E1 -2447.03,E2 -2447.03} C_VEL
LIN {X 0,Y 566.866,Z 342.441,A -85,B 0,C 180,E1 -2449.933,E2 -2449.933} C_VEL
LIN {X 0,Y 566.998,Z 328.459,A -85,B 0,C 180,E1 -2452.02,E2 -2452.02} C_VEL
LIN {X 0,Y 566.183,Z 323.588,A -85,B 0,C 180,E1 -2452.812,E2 -2452.812} C_VEL
LIN {X 0,Y 566.177,Z 323.581,A -85,B 0,C 180,E1 -2455.749,E2 -2455.749} C_VEL
LIN {X 0,Y 566.144,Z 323.585,A -85,B 0,C 180,E1 -2458.19,E2 -2458.19} C_VEL
LIN {X 0,Y 566.173,Z 323.589,A -85,B 0,C 180,E1 -2461.073,E2 -2461.073} C_VEL
LIN {X 0,Y 566.19,Z 323.579,A -85,B 0,C 180,E1 -2463.73,E2 -2463.73} C_VEL
LIN {X 0,Y 566.17,Z 323.585,A -85,B 0,C 180,E1 -2466.57,E2 -2466.57} C_VEL
LIN {X 0,Y 566.197,Z 323.577,A -85,B 0,C 180,E1 -2469.683,E2 -2469.683} C_VEL
LIN {X 0,Y 566.137,Z 323.584,A -85,B 0,C 180,E1 -2472.092,E2 -2472.092} C_VEL
LIN {X 0,Y 566.154,Z 323.589,A -85,B 0,C 180,E1 -2475.036,E2 -2475.036} C_VEL
LIN {X 0,Y 566.157,Z 323.581,A -85,B 0,C 180,E1 -2477.907,E2 -2477.907} C_VEL
LIN {X 0,Y 566.193,Z 323.585,A -85,B 0,C 180,E1 -2480.724,E2 -2480.724} C_VEL
LIN {X 0,Y 566.166,Z 323.582,A -85,B 0,C 180,E1 -2483.427,E2 -2483.427} C_VEL
LIN {X 0,Y 566.183,Z 323.58,A -85,B 0,C 180,E1 -2486.267,E2 -2486.267} C_VEL
LIN {X 0,Y 566.167,Z 323.588,A -85,B 0,C 180,E1 -2488.924,E2 -2488.924} C_VEL
LIN {X 0,Y 566.135,Z 323.583,A -85,B 0,C 180,E1 -2491.853,E2 -2491.853} C_VEL
LIN {X 0,Y 566.174,Z 323.579,A -85,B 0,C 180,E1 -2494.249,E2 -2494.249} C_VEL
LIN {X 0,Y 566.146,Z 323.584,A -85,B 0,C 180,E1 -2497.367,E2 -2497.367} C_VEL
LIN {X 0,Y 566.183,Z 323.576,A -85,B 0,C 180,E1 -2499.662,E2 -2499.662} C_VEL
LIN {X 0,Y 566.157,Z 323.579,A -85,B 0,C 180,E1 -2501.92,E2 -2501.92} C_VEL
LIN {X 0,Y 566.163,Z 323.583,A -85,B 0,C 180,E1 -2504.151,E2 -2504.151} C_VEL
LIN {X 0,Y 566.146,Z 323.588,A -85,B 0,C 180,E1 -2506.358,E2 -2506.358} C_VEL
LIN {X 0,Y 566.199,Z 323.577,A -85,B 0,C 180,E1 -2509.269,E2 -2509.269} C_VEL
LIN {X 0,Y 566.199,Z 323.578,A -85,B 0,C 180,E1 -2512.152,E2 -2512.152} C_VEL
LIN {X 0,Y 566.241,Z 323.573,A -85,B 0,C 180,E1 -2515.016,E2 -2515.016} C_VEL
LIN {X 0,Y 566.243,Z 323.572,A -85,B 0,C 180,E1 -2517.866,E2 -2517.866} C_VEL
LIN {X 0,Y 566.285,Z 323.573,A -85,B 0,C 180,E1 -2520.711,E2 -2520.711} C_VEL
LIN {X 0,Y 566.245,Z 323.575,A -85,B 0,C 180,E1 -2522.846,E2 -2522.846} C_VEL
LIN {X 0,Y 566.214,Z 323.574,A -85,B 0,C 180,E1 -2525.699,E2 -2525.699} C_VEL
LIN {X 0,Y 566.173,Z 323.588,A -85,B 0,C 180,E1 -2528.567,E2 -2528.567} C_VEL
LIN {X 0,Y 566.177,Z 323.579,A -85,B 0,C 180,E1 -2531.456,E2 -2531.456} C_VEL
LIN {X 0,Y 566.214,Z 323.584,A -85,B 0,C 180,E1 -2534.505,E2 -2534.505} C_VEL
LIN {X 0,Y 566.157,Z 323.581,A -85,B 0,C 180,E1 -2537.333,E2 -2537.333} C_VEL
LIN {X 0,Y 566.184,Z 323.578,A -85,B 0,C 180,E1 -2539.582,E2 -2539.582} C_VEL
LIN {X 0,Y 566.173,Z 323.579,A -85,B 0,C 180,E1 -2541.863,E2 -2541.863} C_VEL
LIN {X 0,Y 566.163,Z 323.582,A -85,B 0,C 180,E1 -2545.022,E2 -2545.022} C_VEL
LIN {X 0,Y 566.148,Z 323.582,A -85,B 0,C 180,E1 -2547.342,E2 -2547.342} C_VEL
LIN {X 0,Y 566.151,Z 323.582,A -85,B 0,C 180,E1 -2549.772,E2 -2549.772} C_VEL
LIN {X 0,Y 566.18,Z 323.587,A -85,B 0,C 180,E1 -2552.429,E2 -2552.429} C_VEL
LIN {X 0,Y 566.147,Z 323.584,A -85,B 0,C 180,E1 -2554.987,E2 -2554.987} C_VEL
LIN {X 0,Y 566.17,Z 323.58,A -85,B 0,C 180,E1 -2557.463,E2 -2557.463} C_VEL
LIN {X 0,Y 566.165,Z 323.589,A -85,B 0,C 180,E1 -2560.203,E2 -2560.203} C_VEL
LIN {X 0,Y 566.166,Z 323.581,A -85,B 0,C 180,E1 -2563.058,E2 -2563.058} C_VEL
LIN {X 0,Y 566.132,Z 323.592,A -85,B 0,C 180,E1 -2566.056,E2 -2566.056} C_VEL
LIN {X 0,Y 566.125,Z 323.587,A -85,B 0,C 180,E1 -2568.858,E2 -2568.858} C_VEL
LIN {X 0,Y 566.15,Z 323.585,A -85,B 0,C 180,E1 -2571.636,E2 -2571.636} C_VEL
LIN {X 0,Y 566.127,Z 323.594,A -85,B 0,C 180,E1 -2574.307,E2 -2574.307} C_VEL
LIN {X 0,Y 566.153,Z 323.583,A -85,B 0,C 180,E1 -2576.895,E2 -2576.895} C_VEL
LIN {X 0,Y 566.157,Z 323.582,A -85,B 0,C 180,E1 -2579.407,E2 -2579.407} C_VEL
LIN {X 0,Y 566.131,Z 323.59,A -85,B 0,C 180,E1 -2581.855,E2 -2581.855} C_VEL
LIN {X 0,Y 566.168,Z 323.589,A -85,B 0,C 180,E1 -2584.25,E2 -2584.25} C_VEL
LIN {X 0,Y 566.205,Z 323.763,A -85,B 0,C 180,E1 -2586.211,E2 -2586.211} C_VEL
LIN {X 0,Y 567.132,Z 329.159,A -85,B 0,C 180,E1 -2587.025,E2 -2587.025} C_VEL
LIN {X 0,Y 566.98,Z 345.308,A -85,B 0,C 180,E1 -2589.314,E2 -2589.314} C_VEL
LIN {X 0,Y 566.709,Z 364.106,A -85,B 0,C 180,E1 -2591.94,E2 -2591.94} C_VEL
LIN {X 0,Y 566.657,Z 372.046,A -85,B 0,C 180,E1 -2593.031,E2 -2593.031} C_VEL
LIN {X 0,Y 567.772,Z 378.933,A -85,B 0,C 180,E1 -2593.155,E2 -2593.155} C_VEL
LIN {X 0,Y 567.454,Z 508.712,A -85,B 0,C 180,E1 -2594.834,E2 -2594.834} C_VEL
LIN {X 0,Y 567.3,Z 523.188,A -85,B 0,C 180,E1 -2595.16,E2 -2595.16} C_VEL
LIN {X 0,Y 567.188,Z 536.42,A -85,B 0,C 180,E1 -2595.6,E2 -2595.6} C_VEL
LIN {X 0,Y 566.994,Z 549.901,A -85,B 0,C 180,E1 -2596.197,E2 -2596.197} C_VEL
LIN {X 0,Y 566.797,Z 562.7,A -85,B 0,C 180,E1 -2596.922,E2 -2596.922} C_VEL
LIN {X 0,Y 566.62,Z 574.328,A -85,B 0,C 180,E1 -2597.738,E2 -2597.738} C_VEL
LIN {X 0,Y 566.441,Z 584.234,A -85,B 0,C 180,E1 -2598.573,E2 -2598.573} C_VEL
LIN {X 0,Y 566.294,Z 594.718,A -85,B 0,C 180,E1 -2599.634,E2 -2599.634} C_VEL
LIN {X 0,Y 566.18,Z 603.567,A -85,B 0,C 180,E1 -2600.715,E2 -2600.715} C_VEL
LIN {X 0,Y 566.046,Z 612.044,A -85,B 0,C 180,E1 -2601.972,E2 -2601.972} C_VEL
LIN {X 0,Y 565.965,Z 619.806,A -85,B 0,C 180,E1 -2603.423,E2 -2603.423} C_VEL
LIN {X 0,Y 565.928,Z 624.964,A -85,B 0,C 180,E1 -2604.657,E2 -2604.657} C_VEL
LIN {X 0,Y 565.956,Z 628.449,A -85,B 0,C 180,E1 -2605.728,E2 -2605.728} C_VEL
LIN {X 0,Y 565.874,Z 631.836,A -85,B 0,C 180,E1 -2607.154,E2 -2607.154} C_VEL
LIN {X 0,Y 565.84,Z 633.835,A -85,B 0,C 180,E1 -2608.578,E2 -2608.578} C_VEL
LIN {X 0,Y 565.837,Z 634.5,A -85,B 0,C 180,E1 -2610.001,E2 -2610.001} C_VEL
LIN {X 0,Y 565.84,Z 633.832,A -85,B 0,C 180,E1 -2611.424,E2 -2611.424} C_VEL
LIN {X 0,Y 565.875,Z 631.83,A -85,B 0,C 180,E1 -2612.849,E2 -2612.849} C_VEL
LIN {X 0,Y 565.956,Z 628.44,A -85,B 0,C 180,E1 -2614.274,E2 -2614.274} C_VEL
LIN {X 0,Y 565.983,Z 623.565,A -85,B 0,C 180,E1 -2615.702,E2 -2615.702} C_VEL
LIN {X 0,Y 565.994,Z 619.04,A -85,B 0,C 180,E1 -2616.74,E2 -2616.74} C_VEL
LIN {X 0,Y 566.048,Z 612.03,A -85,B 0,C 180,E1 -2618.03,E2 -2618.03} C_VEL
LIN {X 0,Y 566.178,Z 603.551,A -85,B 0,C 180,E1 -2619.287,E2 -2619.287} C_VEL
LIN {X 0,Y 566.295,Z 594.698,A -85,B 0,C 180,E1 -2620.368,E2 -2620.368} C_VEL
LIN {X 0,Y 566.487,Z 583.979,A -85,B 0,C 180,E1 -2621.45,E2 -2621.45} C_VEL
LIN {X 0,Y 566.609,Z 573.127,A -85,B 0,C 180,E1 -2622.356,E2 -2622.356} C_VEL
LIN {X 0,Y 566.78,Z 561.238,A -85,B 0,C 180,E1 -2623.171,E2 -2623.171} C_VEL
LIN {X 0,Y 567.046,Z 548.078,A -85,B 0,C 180,E1 -2623.895,E2 -2623.895} C_VEL
LIN {X 0,Y 567.228,Z 535.035,A -85,B 0,C 180,E1 -2624.454,E2 -2624.454} C_VEL
LIN {X 0,Y 567.352,Z 521.184,A -85,B 0,C 180,E1 -2624.893,E2 -2624.893} C_VEL
LIN {X 0,Y 567.458,Z 507.07,A -85,B 0,C 180,E1 -2625.191,E2 -2625.191} C_VEL
LIN {X 0,Y 567.688,Z 377.514,A -85,B 0,C 180,E1 -2626.866,E2 -2626.866} C_VEL
LIN {X 0,Y 566.638,Z 371.917,A -85,B 0,C 180,E1 -2626.979,E2 -2626.979} C_VEL
LIN {X 0,Y 566.905,Z 350.665,A -85,B 0,C 180,E1 -2629.934,E2 -2629.934} C_VEL
LIN {X 0,Y 567.222,Z 330.491,A -85,B 0,C 180,E1 -2632.781,E2 -2632.781} C_VEL
LIN {X 0,Y 566.52,Z 325.23,A -85,B 0,C 180,E1 -2633.564,E2 -2633.564} C_VEL
LIN {X 0,Y 566.171,Z 323.59,A -85,B 0,C 180,E1 -2633.842,E2 -2633.842} C_VEL
LIN {X 0,Y 566.17,Z 323.582,A -85,B 0,C 180,E1 -2636.651,E2 -2636.651} C_VEL
LIN {X 0,Y 566.163,Z 323.588,A -85,B 0,C 180,E1 -2639.772,E2 -2639.772} C_VEL
LIN {X 0,Y 566.197,Z 323.578,A -85,B 0,C 180,E1 -2642.429,E2 -2642.429} C_VEL
LIN {X 0,Y 566.18,Z 323.584,A -85,B 0,C 180,E1 -2644.989,E2 -2644.989} C_VEL
LIN {X 0,Y 566.196,Z 323.582,A -85,B 0,C 180,E1 -2647.462,E2 -2647.462} C_VEL
LIN {X 0,Y 566.214,Z 323.575,A -85,B 0,C 180,E1 -2650.199,E2 -2650.199} C_VEL
LIN {X 0,Y 566.204,Z 323.584,A -85,B 0,C 180,E1 -2653.055,E2 -2653.055} C_VEL
LIN {X 0,Y 566.203,Z 323.577,A -85,B 0,C 180,E1 -2656.049,E2 -2656.049} C_VEL
LIN {X 0,Y 566.209,Z 323.578,A -85,B 0,C 180,E1 -2659.215,E2 -2659.215} C_VEL
LIN {X 0,Y 566.187,Z 323.579,A -85,B 0,C 180,E1 -2661.637,E2 -2661.637} C_VEL
LIN {X 0,Y 566.155,Z 323.59,A -85,B 0,C 180,E1 -2664.307,E2 -2664.307} C_VEL
LIN {X 0,Y 566.224,Z 323.576,A -85,B 0,C 180,E1 -2666.898,E2 -2666.898} C_VEL
LIN {X 0,Y 566.181,Z 323.581,A -85,B 0,C 180,E1 -2669.407,E2 -2669.407} C_VEL
LIN {X 0,Y 566.191,Z 323.587,A -85,B 0,C 180,E1 -2671.856,E2 -2671.856} C_VEL
LIN {X 0,Y 566.187,Z 323.584,A -85,B 0,C 180,E1 -2674.25,E2 -2674.25} C_VEL
LIN {X 0,Y 566.17,Z 323.584,A -85,B 0,C 180,E1 -2676.72,E2 -2676.72} C_VEL
LIN {X 0,Y 566.21,Z 323.675,A -85,B 0,C 180,E1 -2678.222,E2 -2678.222} C_VEL
LIN {X 0,Y 566.798,Z 329.238,A -85,B 0,C 180,E1 -2679.116,E2 -2679.116} C_VEL
LIN {X 0,Y 566.602,Z 345.812,A -85,B 0,C 180,E1 -2681.748,E2 -2681.748} C_VEL
LIN {X 0,Y 566.396,Z 363.314,A -85,B 0,C 180,E1 -2684.527,E2 -2684.527} C_VEL
LIN {X 0,Y 566.356,Z 372.94,A -85,B 0,C 180,E1 -2686.042,E2 -2686.042} C_VEL
LIN {X 0,Y 567.17,Z 378.064,A -85,B 0,C 180,E1 -2686.131,E2 -2686.131} C_VEL
LIN {X 0,Y 566.942,Z 480.376,A -85,B 0,C 180,E1 -2687.448,E2 -2687.448} C_VEL
LIN {X 0,Y 566.877,Z 493.741,A -85,B 0,C 180,E1 -2687.765,E2 -2687.765} C_VEL
LIN {X 0,Y 566.754,Z 505.869,A -85,B 0,C 180,E1 -2688.194,E2 -2688.194} C_VEL
LIN {X 0,Y 566.635,Z 517.957,A -85,B 0,C 180,E1 -2688.77,E2 -2688.77} C_VEL
LIN {X 0,Y 566.461,Z 529.061,A -85,B 0,C 180,E1 -2689.455,E2 -2689.455} C_VEL
LIN {X 0,Y 566.316,Z 539.551,A -85,B 0,C 180,E1 -2690.265,E2 -2690.265} C_VEL
LIN {X 0,Y 566.212,Z 548.17,A -85,B 0,C 180,E1 -2691.074,E2 -2691.074} C_VEL
LIN {X 0,Y 566.095,Z 557.472,A -85,B 0,C 180,E1 -2692.151,E2 -2692.151} C_VEL
LIN {X 0,Y 566.019,Z 564.35,A -85,B 0,C 180,E1 -2693.127,E2 -2693.127} C_VEL
LIN {X 0,Y 566.004,Z 570.944,A -85,B 0,C 180,E1 -2694.299,E2 -2694.299} C_VEL
LIN {X 0,Y 565.933,Z 575.709,A -85,B 0,C 180,E1 -2695.37,E2 -2695.37} C_VEL
LIN {X 0,Y 565.928,Z 579.308,A -85,B 0,C 180,E1 -2696.44,E2 -2696.44} C_VEL
LIN {X 0,Y 565.878,Z 581.175,A -85,B 0,C 180,E1 -2697.153,E2 -2697.153} C_VEL
LIN {X 0,Y 565.846,Z 583.638,A -85,B 0,C 180,E1 -2698.577,E2 -2698.577} C_VEL
LIN {X 0,Y 565.841,Z 584.268,A -85,B 0,C 180,E1 -2699.288,E2 -2699.288} C_VEL
LIN {X 0,Y 565.839,Z 584.496,A -85,B 0,C 180,E1 -2700,E2 -2700} C_VEL
LIN {X 0,Y 565.841,Z 584.318,A -85,B 0,C 180,E1 -2700.712,E2 -2700.712} C_VEL
LIN {X 0,Y 565.846,Z 583.734,A -85,B 0,C 180,E1 -2701.423,E2 -2701.423} C_VEL
LIN {X 0,Y 565.879,Z 581.379,A -85,B 0,C 180,E1 -2702.848,E2 -2702.848} C_VEL
LIN {X 0,Y 565.927,Z 578.522,A -85,B 0,C 180,E1 -2703.917,E2 -2703.917} C_VEL
LIN {X 0,Y 565.878,Z 574.63,A -85,B 0,C 180,E1 -2704.988,E2 -2704.988} C_VEL
LIN {X 0,Y 565.988,Z 569.572,A -85,B 0,C 180,E1 -2706.059,E2 -2706.059} C_VEL
LIN {X 0,Y 566.032,Z 563.255,A -85,B 0,C 180,E1 -2707.132,E2 -2707.132} C_VEL
LIN {X 0,Y 566.128,Z 555.364,A -85,B 0,C 180,E1 -2708.208,E2 -2708.208} C_VEL
LIN {X 0,Y 566.206,Z 547.273,A -85,B 0,C 180,E1 -2709.106,E2 -2709.106} C_VEL
LIN {X 0,Y 566.333,Z 537.44,A -85,B 0,C 180,E1 -2710.005,E2 -2710.005} C_VEL
LIN {X 0,Y 566.508,Z 526.465,A -85,B 0,C 180,E1 -2710.807,E2 -2710.807} C_VEL
LIN {X 0,Y 566.615,Z 515.535,A -85,B 0,C 180,E1 -2711.447,E2 -2711.447} C_VEL
LIN {X 0,Y 566.764,Z 502.792,A -85,B 0,C 180,E1 -2712.02,E2 -2712.02} C_VEL
LIN {X 0,Y 566.91,Z 489.706,A -85,B 0,C 180,E1 -2712.439,E2 -2712.439} C_VEL
LIN {X 0,Y 567.006,Z 476.144,A -85,B 0,C 180,E1 -2712.71,E2 -2712.71} C_VEL
LIN {X 0,Y 567.217,Z 380.817,A -85,B 0,C 180,E1 -2713.922,E2 -2713.922} C_VEL
LIN {X 0,Y 566.855,Z 377.195,A -85,B 0,C 180,E1 -2714.029,E2 -2714.029} C_VEL
LIN {X 0,Y 565.93,Z 374.009,A -85,B 0,C 180,E1 -2714.223,E2 -2714.223} C_VEL
LIN {X 0,Y 563.994,Z 370.019,A -85,B 0,C 180,E1 -2714.621,E2 -2714.621} C_VEL
LIN {X 0,Y 561.874,Z 366.946,A -85,B 0,C 180,E1 -2715.113,E2 -2715.113} C_VEL
LIN {X 0,Y 559.762,Z 362.788,A -85,B 0,C 180,E1 -2715.839,E2 -2715.839} C_VEL
LIN {X 0,Y 559.459,Z 360.523,A -85,B 0,C 180,E1 -2716.207,E2 -2716.207} C_VEL
LIN {X 0,Y 559.656,Z 342.78,A -85,B 0,C 180,E1 -2719.057,E2 -2719.057} C_VEL
LIN {X 0,Y 559.817,Z 329.8,A -85,B 0,C 180,E1 -2721.157,E2 -2721.157} C_VEL
LIN {X 0,Y 559.196,Z 324.458,A -85,B 0,C 180,E1 -2722.042,E2 -2722.042} C_VEL
LIN {X 0,Y 559.181,Z 324.452,A -85,B 0,C 180,E1 -2725.298,E2 -2725.298} C_VEL
LIN {X 0,Y 559.145,Z 324.459,A -85,B 0,C 180,E1 -2727.714,E2 -2727.714} C_VEL
LIN {X 0,Y 559.157,Z 324.462,A -85,B 0,C 180,E1 -2730.183,E2 -2730.183} C_VEL
LIN {X 0,Y 559.161,Z 324.455,A -85,B 0,C 180,E1 -2732.715,E2 -2732.715} C_VEL
LIN {X 0,Y 559.127,Z 324.459,A -85,B 0,C 180,E1 -2735.324,E2 -2735.324} C_VEL
LIN {X 0,Y 559.134,Z 324.465,A -85,B 0,C 180,E1 -2738.018,E2 -2738.018} C_VEL
LIN {X 0,Y 559.159,Z 324.453,A -85,B 0,C 180,E1 -2740.812,E2 -2740.812} C_VEL
LIN {X 0,Y 559.141,Z 324.465,A -85,B 0,C 180,E1 -2743.734,E2 -2743.734} C_VEL
LIN {X 0,Y 559.135,Z 324.457,A -85,B 0,C 180,E1 -2746.805,E2 -2746.805} C_VEL
LIN {X 0,Y 559.131,Z 324.461,A -85,B 0,C 180,E1 -2749.185,E2 -2749.185} C_VEL
LIN {X 0,Y 559.127,Z 324.461,A -85,B 0,C 180,E1 -2751.981,E2 -2751.981} C_VEL
LIN {X 0,Y 559.127,Z 324.459,A -85,B 0,C 180,E1 -2754.788,E2 -2754.788} C_VEL
LIN {X 0,Y 559.143,Z 324.464,A -85,B 0,C 180,E1 -2757.367,E2 -2757.367} C_VEL
LIN {X 0,Y 559.11,Z 324.461,A -85,B 0,C 180,E1 -2760.15,E2 -2760.15} C_VEL
LIN {X 0,Y 559.11,Z 324.466,A -85,B 0,C 180,E1 -2763.185,E2 -2763.185} C_VEL
LIN {X 0,Y 559.087,Z 324.47,A -85,B 0,C 180,E1 -2765.491,E2 -2765.491} C_VEL
LIN {X 0,Y 559.164,Z 324.583,A -85,B 0,C 180,E1 -2767.141,E2 -2767.141} C_VEL
LIN {X 0,Y 560.123,Z 330.63,A -85,B 0,C 180,E1 -2768.111,E2 -2768.111} C_VEL
LIN {X 0,Y 559.804,Z 348.391,A -85,B 0,C 180,E1 -2770.788,E2 -2770.788} C_VEL
LIN {X 0,Y 559.629,Z 362.298,A -85,B 0,C 180,E1 -2772.852,E2 -2772.852} C_VEL
LIN {X 0,Y 561.024,Z 370.757,A -85,B 0,C 180,E1 -2773.015,E2 -2773.015} C_VEL
LIN {X 0,Y 560.565,Z 498.23,A -85,B 0,C 180,E1 -2774.688,E2 -2774.688} C_VEL
LIN {X 0,Y 560.442,Z 510.155,A -85,B 0,C 180,E1 -2774.943,E2 -2774.943} C_VEL
LIN {X 0,Y 560.356,Z 522.538,A -85,B 0,C 180,E1 -2775.323,E2 -2775.323} C_VEL
LIN {X 0,Y 560.174,Z 535.203,A -85,B 0,C 180,E1 -2775.838,E2 -2775.838} C_VEL
LIN {X 0,Y 559.879,Z 548.962,A -85,B 0,C 180,E1 -2776.571,E2 -2776.571} C_VEL
LIN {X 0,Y 559.707,Z 560.004,A -85,B 0,C 180,E1 -2777.305,E2 -2777.305} C_VEL
LIN {X 0,Y 559.531,Z 569.289,A -85,B 0,C 180,E1 -2778.038,E2 -2778.038} C_VEL
LIN {X 0,Y 559.42,Z 578.256,A -85,B 0,C 180,E1 -2778.867,E2 -2778.867} C_VEL
LIN {X 0,Y 559.24,Z 585.864,A -85,B 0,C 180,E1 -2779.683,E2 -2779.683} C_VEL
LIN {X 0,Y 559.122,Z 593.178,A -85,B 0,C 180,E1 -2780.594,E2 -2780.594} C_VEL
LIN {X 0,Y 559.008,Z 600.591,A -85,B 0,C 180,E1 -2781.686,E2 -2781.686} C_VEL
LIN {X 0,Y 558.909,Z 606.78,A -85,B 0,C 180,E1 -2782.775,E2 -2782.775} C_VEL
LIN {X 0,Y 558.887,Z 611.879,A -85,B 0,C 180,E1 -2783.863,E2 -2783.863} C_VEL
LIN {X 0,Y 558.821,Z 617.251,A -85,B 0,C 180,E1 -2785.31,E2 -2785.31} C_VEL
LIN {X 0,Y 558.826,Z 620.211,A -85,B 0,C 180,E1 -2786.394,E2 -2786.394} C_VEL
LIN {X 0,Y 558.745,Z 622.944,A -85,B 0,C 180,E1 -2787.836,E2 -2787.836} C_VEL
LIN {X 0,Y 558.737,Z 624.266,A -85,B 0,C 180,E1 -2789.278,E2 -2789.278} C_VEL
LIN {X 0,Y 558.739,Z 624.496,A -85,B 0,C 180,E1 -2789.999,E2 -2789.999} C_VEL
LIN {X 0,Y 558.741,Z 623.855,A -85,B 0,C 180,E1 -2791.44,E2 -2791.44} C_VEL
LIN {X 0,Y 558.794,Z 621.876,A -85,B 0,C 180,E1 -2792.883,E2 -2792.883} C_VEL
LIN {X 0,Y 558.826,Z 620.437,A -85,B 0,C 180,E1 -2793.604,E2 -2793.604} C_VEL
LIN {X 0,Y 558.791,Z 616.33,A -85,B 0,C 180,E1 -2795.05,E2 -2795.05} C_VEL
LIN {X 0,Y 558.883,Z 612.277,A -85,B 0,C 180,E1 -2796.135,E2 -2796.135} C_VEL
LIN {X 0,Y 558.905,Z 607.262,A -85,B 0,C 180,E1 -2797.223,E2 -2797.223} C_VEL
LIN {X 0,Y 559.006,Z 601.164,A -85,B 0,C 180,E1 -2798.312,E2 -2798.312} C_VEL
LIN {X 0,Y 559.105,Z 593.85,A -85,B 0,C 180,E1 -2799.404,E2 -2799.404} C_VEL
LIN {X 0,Y 559.263,Z 585.093,A -85,B 0,C 180,E1 -2800.498,E2 -2800.498} C_VEL
LIN {X 0,Y 559.453,Z 574.512,A -85,B 0,C 180,E1 -2801.594,E2 -2801.594} C_VEL
LIN {X 0,Y 559.629,Z 563.715,A -85,B 0,C 180,E1 -2802.51,E2 -2802.51} C_VEL
LIN {X 0,Y 559.806,Z 553.342,A -85,B 0,C 180,E1 -2803.244,E2 -2803.244} C_VEL
LIN {X 0,Y 560.019,Z 542.406,A -85,B 0,C 180,E1 -2803.886,E2 -2803.886} C_VEL
LIN {X 0,Y 560.176,Z 531.99,A -85,B 0,C 180,E1 -2804.392,E2 -2804.392} C_VEL
LIN {X 0,Y 560.39,Z 520.38,A -85,B 0,C 180,E1 -2804.839,E2 -2804.839} C_VEL
LIN {X 0,Y 560.502,Z 509.102,A -85,B 0,C 180,E1 -2805.172,E2 -2805.172} C_VEL
LIN {X 0,Y 560.57,Z 498.179,A -85,B 0,C 180,E1 -2805.403,E2 -2805.403} C_VEL
LIN {X 0,Y 560.93,Z 369.35,A -85,B 0,C 180,E1 -2807.096,E2 -2807.096} C_VEL
LIN {X 0,Y 559.624,Z 362.309,A -85,B 0,C 180,E1 -2807.236,E2 -2807.236} C_VEL
LIN {X 0,Y 559.95,Z 341.19,A -85,B 0,C 180,E1 -2810.382,E2 -2810.382} C_VEL
LIN {X 0,Y 560.068,Z 329.785,A -85,B 0,C 180,E1 -2812.113,E2 -2812.113} C_VEL
LIN {X 0,Y 559.152,Z 324.464,A -85,B 0,C 180,E1 -2813.003,E2 -2813.003} C_VEL
LIN {X 0,Y 559.143,Z 324.457,A -85,B 0,C 180,E1 -2816.097,E2 -2816.097} C_VEL
LIN {X 0,Y 559.103,Z 324.465,A -85,B 0,C 180,E1 -2818.531,E2 -2818.531} C_VEL
LIN {X 0,Y 559.129,Z 324.464,A -85,B 0,C 180,E1 -2821.27,E2 -2821.27} C_VEL
LIN {X 0,Y 559.147,Z 324.456,A -85,B 0,C 180,E1 -2823.946,E2 -2823.946} C_VEL
LIN {X 0,Y 559.118,Z 324.466,A -85,B 0,C 180,E1 -2827.108,E2 -2827.108} C_VEL
LIN {X 0,Y 559.146,Z 324.455,A -85,B 0,C 180,E1 -2829.94,E2 -2829.94} C_VEL
LIN {X 0,Y 559.114,Z 324.464,A -85,B 0,C 180,E1 -2833.193,E2 -2833.193} C_VEL
LIN {X 0,Y 559.118,Z 324.458,A -85,B 0,C 180,E1 -2835.762,E2 -2835.762} C_VEL
LIN {X 0,Y 559.111,Z 324.461,A -85,B 0,C 180,E1 -2838.225,E2 -2838.225} C_VEL
LIN {X 0,Y 559.155,Z 324.456,A -85,B 0,C 180,E1 -2841.192,E2 -2841.192} C_VEL
LIN {X 0,Y 559.104,Z 324.46,A -85,B 0,C 180,E1 -2843.786,E2 -2843.786} C_VEL
LIN {X 0,Y 559.131,Z 324.46,A -85,B 0,C 180,E1 -2846.423,E2 -2846.423} C_VEL
LIN {X 0,Y 559.132,Z 324.463,A -85,B 0,C 180,E1 -2848.979,E2 -2848.979} C_VEL
LIN {X 0,Y 559.096,Z 324.46,A -85,B 0,C 180,E1 -2851.629,E2 -2851.629} C_VEL
LIN {X 0,Y 559.141,Z 324.452,A -85,B 0,C 180,E1 -2853.901,E2 -2853.901} C_VEL
LIN {X 0,Y 559.096,Z 324.465,A -85,B 0,C 180,E1 -2857.065,E2 -2857.065} C_VEL
LIN {X 0,Y 559.155,Z 324.452,A -85,B 0,C 180,E1 -2859.394,E2 -2859.394} C_VEL
LIN {X 0,Y 559.106,Z 324.457,A -85,B 0,C 180,E1 -2861.684,E2 -2861.684} C_VEL
LIN {X 0,Y 559.124,Z 324.458,A -85,B 0,C 180,E1 -2863.947,E2 -2863.947} C_VEL
LIN {X 0,Y 559.126,Z 324.46,A -85,B 0,C 180,E1 -2866.183,E2 -2866.183} C_VEL
LIN {X 0,Y 559.162,Z 324.455,A -85,B 0,C 180,E1 -2869.133,E2 -2869.133} C_VEL
LIN {X 0,Y 559.169,Z 324.453,A -85,B 0,C 180,E1 -2872.053,E2 -2872.053} C_VEL
LIN {X 0,Y 559.217,Z 324.449,A -85,B 0,C 180,E1 -2874.953,E2 -2874.953} C_VEL
LIN {X 0,Y 559.216,Z 324.447,A -85,B 0,C 180,E1 -2877.839,E2 -2877.839} C_VEL
LIN {X 0,Y 559.255,Z 324.448,A -85,B 0,C 180,E1 -2880.72,E2 -2880.72} C_VEL
LIN {X 0,Y 559.21,Z 324.451,A -85,B 0,C 180,E1 -2882.881,E2 -2882.881} C_VEL
LIN {X 0,Y 559.185,Z 324.45,A -85,B 0,C 180,E1 -2885.771,E2 -2885.771} C_VEL
LIN {X 0,Y 559.139,Z 324.462,A -85,B 0,C 180,E1 -2888.675,E2 -2888.675} C_VEL
LIN {X 0,Y 559.143,Z 324.455,A -85,B 0,C 180,E1 -2891.602,E2 -2891.602} C_VEL
LIN {X 0,Y 559.185,Z 324.458,A -85,B 0,C 180,E1 -2894.596,E2 -2894.596} C_VEL
LIN {X 0,Y 559.107,Z 324.459,A -85,B 0,C 180,E1 -2897.559,E2 -2897.559} C_VEL
LIN {X 0,Y 559.148,Z 324.456,A -85,B 0,C 180,E1 -2899.838,E2 -2899.838} C_VEL
LIN {X 0,Y 559.118,Z 324.461,A -85,B 0,C 180,E1 -2902.154,E2 -2902.154} C_VEL
LIN {X 0,Y 559.122,Z 324.458,A -85,B 0,C 180,E1 -2905.178,E2 -2905.178} C_VEL
LIN {X 0,Y 559.118,Z 324.465,A -85,B 0,C 180,E1 -2908.375,E2 -2908.375} C_VEL
LIN {X 0,Y 559.109,Z 324.459,A -85,B 0,C 180,E1 -2911.27,E2 -2911.27} C_VEL
LIN {X 0,Y 559.137,Z 324.459,A -85,B 0,C 180,E1 -2913.948,E2 -2913.948} C_VEL
LIN {X 0,Y 559.098,Z 324.461,A -85,B 0,C 180,E1 -2917.112,E2 -2917.112} C_VEL
LIN {X 0,Y 559.138,Z 324.459,A -85,B 0,C 180,E1 -2919.869,E2 -2919.869} C_VEL
LIN {X 0,Y 559.111,Z 324.459,A -85,B 0,C 180,E1 -2923.195,E2 -2923.195} C_VEL
LIN {X 0,Y 559.102,Z 324.464,A -85,B 0,C 180,E1 -2925.766,E2 -2925.766} C_VEL
LIN {X 0,Y 559.083,Z 324.473,A -85,B 0,C 180,E1 -2928.224,E2 -2928.224} C_VEL
LIN {X 0,Y 559.126,Z 324.458,A -85,B 0,C 180,E1 -2931.198,E2 -2931.198} C_VEL
LIN {X 0,Y 559.102,Z 324.465,A -85,B 0,C 180,E1 -2933.788,E2 -2933.788} C_VEL
LIN {X 0,Y 559.127,Z 324.464,A -85,B 0,C 180,E1 -2936.424,E2 -2936.424} C_VEL
LIN {X 0,Y 559.139,Z 324.456,A -85,B 0,C 180,E1 -2938.981,E2 -2938.981} C_VEL
LIN {X 0,Y 559.094,Z 324.464,A -85,B 0,C 180,E1 -2941.633,E2 -2941.633} C_VEL
LIN {X 0,Y 559.136,Z 324.464,A -85,B 0,C 180,E1 -2943.902,E2 -2943.902} C_VEL
LIN {X 0,Y 559.138,Z 324.54,A -85,B 0,C 180,E1 -2946.014,E2 -2946.014} C_VEL
LIN {X 0,Y 560.252,Z 330.617,A -85,B 0,C 180,E1 -2946.946,E2 -2946.946} C_VEL
LIN {X 0,Y 560.066,Z 347.973,A -85,B 0,C 180,E1 -2949.431,E2 -2949.431} C_VEL
LIN {X 0,Y 559.704,Z 370.55,A -85,B 0,C 180,E1 -2952.613,E2 -2952.613} C_VEL
LIN {X 0,Y 559.732,Z 372.095,A -85,B 0,C 180,E1 -2952.816,E2 -2952.816} C_VEL
LIN {X 0,Y 560.964,Z 379.069,A -85,B 0,C 180,E1 -2952.946,E2 -2952.946} C_VEL
LIN {X 0,Y 560.609,Z 508.712,A -85,B 0,C 180,E1 -2954.644,E2 -2954.644} C_VEL
LIN {X 0,Y 560.472,Z 522.737,A -85,B 0,C 180,E1 -2954.962,E2 -2954.962} C_VEL
LIN {X 0,Y 560.314,Z 536.512,A -85,B 0,C 180,E1 -2955.423,E2 -2955.423} C_VEL
LIN {X 0,Y 560.086,Z 549.899,A -85,B 0,C 180,E1 -2956.023,E2 -2956.023} C_VEL
LIN {X 0,Y 559.841,Z 562.698,A -85,B 0,C 180,E1 -2956.757,E2 -2956.757} C_VEL
LIN {X 0,Y 559.647,Z 574.326,A -85,B 0,C 180,E1 -2957.583,E2 -2957.583} C_VEL
LIN {X 0,Y 559.429,Z 584.93,A -85,B 0,C 180,E1 -2958.493,E2 -2958.493} C_VEL
LIN {X 0,Y 559.272,Z 594.718,A -85,B 0,C 180,E1 -2959.503,E2 -2959.503} C_VEL
LIN {X 0,Y 559.12,Z 603.566,A -85,B 0,C 180,E1 -2960.597,E2 -2960.597} C_VEL
LIN {X 0,Y 558.985,Z 612.043,A -85,B 0,C 180,E1 -2961.87,E2 -2961.87} C_VEL
LIN {X 0,Y 558.9,Z 618.87,A -85,B 0,C 180,E1 -2963.141,E2 -2963.141} C_VEL
LIN {X 0,Y 558.912,Z 623.572,A -85,B 0,C 180,E1 -2964.228,E2 -2964.228} C_VEL
LIN {X 0,Y 558.865,Z 628.449,A -85,B 0,C 180,E1 -2965.674,E2 -2965.674} C_VEL
LIN {X 0,Y 558.796,Z 631.837,A -85,B 0,C 180,E1 -2967.117,E2 -2967.117} C_VEL
LIN {X 0,Y 558.74,Z 633.836,A -85,B 0,C 180,E1 -2968.56,E2 -2968.56} C_VEL
LIN {X 0,Y 558.738,Z 634.5,A -85,B 0,C 180,E1 -2970.001,E2 -2970.001} C_VEL
LIN {X 0,Y 558.74,Z 633.832,A -85,B 0,C 180,E1 -2971.443,E2 -2971.443} C_VEL
LIN {X 0,Y 558.796,Z 631.83,A -85,B 0,C 180,E1 -2972.885,E2 -2972.885} C_VEL
LIN {X 0,Y 558.865,Z 628.441,A -85,B 0,C 180,E1 -2974.328,E2 -2974.328} C_VEL
LIN {X 0,Y 558.911,Z 623.565,A -85,B 0,C 180,E1 -2975.774,E2 -2975.774} C_VEL
LIN {X 0,Y 558.903,Z 618.861,A -85,B 0,C 180,E1 -2976.862,E2 -2976.862} C_VEL
LIN {X 0,Y 558.987,Z 612.029,A -85,B 0,C 180,E1 -2978.132,E2 -2978.132} C_VEL
LIN {X 0,Y 559.118,Z 603.55,A -85,B 0,C 180,E1 -2979.406,E2 -2979.406} C_VEL
LIN {X 0,Y 559.273,Z 594.698,A -85,B 0,C 180,E1 -2980.5,E2 -2980.5} C_VEL
LIN {X 0,Y 559.489,Z 583.978,A -85,B 0,C 180,E1 -2981.595,E2 -2981.595} C_VEL
LIN {X 0,Y 559.64,Z 573.125,A -85,B 0,C 180,E1 -2982.512,E2 -2982.512} C_VEL
LIN {X 0,Y 559.855,Z 561.236,A -85,B 0,C 180,E1 -2983.337,E2 -2983.337} C_VEL
LIN {X 0,Y 560.124,Z 548.079,A -85,B 0,C 180,E1 -2984.071,E2 -2984.071} C_VEL
LIN {X 0,Y 560.353,Z 535.239,A -85,B 0,C 180,E1 -2984.627,E2 -2984.627} C_VEL
LIN {X 0,Y 560.496,Z 521.244,A -85,B 0,C 180,E1 -2985.078,E2 -2985.078} C_VEL
LIN {X 0,Y 560.622,Z 507.07,A -85,B 0,C 180,E1 -2985.381,E2 -2985.381} C_VEL
LIN {X 0,Y 560.964,Z 378.917,A -85,B 0,C 180,E1 -2987.056,E2 -2987.056} C_VEL
LIN {X 0,Y 559.687,Z 371.832,A -85,B 0,C 180,E1 -2987.208,E2 -2987.208} C_VEL
LIN {X 0,Y 560.016,Z 349.303,A -85,B 0,C 180,E1 -2990.381,E2 -2990.381} C_VEL
LIN {X 0,Y 560.283,Z 330.608,A -85,B 0,C 180,E1 -2993.054,E2 -2993.054} C_VEL
LIN {X 0,Y 559.14,Z 324.465,A -85,B 0,C 180,E1 -2994.013,E2 -2994.013} C_VEL
LIN {X 0,Y 559.114,Z 324.462,A -85,B 0,C 180,E1 -2996.906,E2 -2996.906} C_VEL
LIN {X 0,Y 559.114,Z 324.465,A -85,B 0,C 180,E1 -2999.851,E2 -2999.851} C_VEL
LIN {X 0,Y 559.155,Z 324.456,A -85,B 0,C 180,E1 -3002.716,E2 -3002.716} C_VEL
LIN {X 0,Y 559.126,Z 324.467,A -85,B 0,C 180,E1 -3005.325,E2 -3005.325} C_VEL
LIN {X 0,Y 559.135,Z 324.457,A -85,B 0,C 180,E1 -3008.018,E2 -3008.018} C_VEL
LIN {X 0,Y 559.16,Z 324.46,A -85,B 0,C 180,E1 -3010.813,E2 -3010.813} C_VEL
LIN {X 0,Y 559.143,Z 324.457,A -85,B 0,C 180,E1 -3013.735,E2 -3013.735} C_VEL
LIN {X 0,Y 559.17,Z 324.461,A -85,B 0,C 180,E1 -3016.802,E2 -3016.802} C_VEL
LIN {X 0,Y 559.16,Z 324.456,A -85,B 0,C 180,E1 -3019.188,E2 -3019.188} C_VEL
LIN {X 0,Y 559.134,Z 324.46,A -85,B 0,C 180,E1 -3021.982,E2 -3021.982} C_VEL
LIN {X 0,Y 559.133,Z 324.461,A -85,B 0,C 180,E1 -3024.788,E2 -3024.788} C_VEL
LIN {X 0,Y 559.16,Z 324.455,A -85,B 0,C 180,E1 -3027.365,E2 -3027.365} C_VEL
LIN {X 0,Y 559.15,Z 324.465,A -85,B 0,C 180,E1 -3030.143,E2 -3030.143} C_VEL
LIN {X 0,Y 559.116,Z 324.462,A -85,B 0,C 180,E1 -3033.095,E2 -3033.095} C_VEL
LIN {X 0,Y 559.126,Z 324.463,A -85,B 0,C 180,E1 -3035.493,E2 -3035.493} C_VEL
LIN {X 0,Y 559.174,Z 324.64,A -85,B 0,C 180,E1 -3038.119,E2 -3038.119} C_VEL
LIN {X 0,Y 559.818,Z 330.167,A -85,B 0,C 180,E1 -3039.035,E2 -3039.035} C_VEL
LIN {X 0,Y 559.585,Z 349.277,A -85,B 0,C 180,E1 -3042.079,E2 -3042.079} C_VEL
LIN {X 0,Y 559.361,Z 366.935,A -85,B 0,C 180,E1 -3044.906,E2 -3044.906} C_VEL
LIN {X 0,Y 559.332,Z 372.944,A -85,B 0,C 180,E1 -3045.864,E2 -3045.864} C_VEL
LIN {X 0,Y 560.306,Z 379.899,A -85,B 0,C 180,E1 -3045.981,E2 -3045.981} C_VEL
LIN {X 0,Y 560.019,Z 480.391,A -85,B 0,C 180,E1 -3047.29,E2 -3047.29} C_VEL
LIN {X 0,Y 559.935,Z 493.753,A -85,B 0,C 180,E1 -3047.611,E2 -3047.611} C_VEL
LIN {X 0,Y 559.812,Z 505.882,A -85,B 0,C 180,E1 -3048.045,E2 -3048.045} C_VEL
LIN {X 0,Y 559.65,Z 517.556,A -85,B 0,C 180,E1 -3048.607,E2 -3048.607} C_VEL
LIN {X 0,Y 559.483,Z 529.06,A -85,B 0,C 180,E1 -3049.322,E2 -3049.322} C_VEL
LIN {X 0,Y 559.298,Z 539.55,A -85,B 0,C 180,E1 -3050.142,E2 -3050.142} C_VEL
LIN {X 0,Y 559.192,Z 548.176,A -85,B 0,C 180,E1 -3050.961,E2 -3050.961} C_VEL
LIN {X 0,Y 559.053,Z 557.47,A -85,B 0,C 180,E1 -3052.051,E2 -3052.051} C_VEL
LIN {X 0,Y 558.932,Z 565.184,A -85,B 0,C 180,E1 -3053.176,E2 -3053.176} C_VEL
LIN {X 0,Y 558.936,Z 570.945,A -85,B 0,C 180,E1 -3054.227,E2 -3054.227} C_VEL
LIN {X 0,Y 558.843,Z 575.712,A -85,B 0,C 180,E1 -3055.311,E2 -3055.311} C_VEL
LIN {X 0,Y 558.837,Z 579.306,A -85,B 0,C 180,E1 -3056.395,E2 -3056.395} C_VEL
LIN {X 0,Y 558.8,Z 581.171,A -85,B 0,C 180,E1 -3057.116,E2 -3057.116} C_VEL
LIN {X 0,Y 558.746,Z 583.639,A -85,B 0,C 180,E1 -3058.559,E2 -3058.559} C_VEL
LIN {X 0,Y 558.742,Z 584.271,A -85,B 0,C 180,E1 -3059.279,E2 -3059.279} C_VEL
LIN {X 0,Y 558.74,Z 584.496,A -85,B 0,C 180,E1 -3060,E2 -3060} C_VEL
LIN {X 0,Y 558.741,Z 584.315,A -85,B 0,C 180,E1 -3060.721,E2 -3060.721} C_VEL
LIN {X 0,Y 558.745,Z 583.729,A -85,B 0,C 180,E1 -3061.442,E2 -3061.442} C_VEL
LIN {X 0,Y 558.8,Z 581.372,A -85,B 0,C 180,E1 -3062.884,E2 -3062.884} C_VEL
LIN {X 0,Y 558.844,Z 578.519,A -85,B 0,C 180,E1 -3063.966,E2 -3063.966} C_VEL
LIN {X 0,Y 558.798,Z 574.623,A -85,B 0,C 180,E1 -3065.051,E2 -3065.051} C_VEL
LIN {X 0,Y 558.908,Z 569.565,A -85,B 0,C 180,E1 -3066.136,E2 -3066.136} C_VEL
LIN {X 0,Y 558.973,Z 563.247,A -85,B 0,C 180,E1 -3067.223,E2 -3067.223} C_VEL
LIN {X 0,Y 559.091,Z 555.356,A -85,B 0,C 180,E1 -3068.312,E2 -3068.312} C_VEL
LIN {X 0,Y 559.173,Z 547.259,A -85,B 0,C 180,E1 -3069.221,E2 -3069.221} C_VEL
LIN {X 0,Y 559.344,Z 537.433,A -85,B 0,C 180,E1 -3070.131,E2 -3070.131} C_VEL
LIN {X 0,Y 559.52,Z 526.546,A -85,B 0,C 180,E1 -3070.937,E2 -3070.937} C_VEL
LIN {X 0,Y 559.666,Z 514.89,A -85,B 0,C 180,E1 -3071.624,E2 -3071.624} C_VEL
LIN {X 0,Y 559.806,Z 502.774,A -85,B 0,C 180,E1 -3072.171,E2 -3072.171} C_VEL
LIN {X 0,Y 559.992,Z 489.69,A -85,B 0,C 180,E1 -3072.595,E2 -3072.595} C_VEL
LIN {X 0,Y 560.078,Z 476.103,A -85,B 0,C 180,E1 -3072.87,E2 -3072.87} C_VEL
LIN {X 0,Y 560.177,Z 378.246,A -85,B 0,C 180,E1 -3074.133,E2 -3074.133} C_VEL
LIN {X 0,Y 559.329,Z 372.926,A -85,B 0,C 180,E1 -3074.229,E2 -3074.229} C_VEL
LIN {X 0,Y 559.459,Z 360.523,A -85,B 0,C 180,E1 -3076.207,E2 -3076.207} C_VEL
LIN {X 0,Y 558.846,Z 357.467,A -85,B 0,C 180,E1 -3076.72,E2 -3076.72} C_VEL
LIN {X 0,Y 553.259,Z 348.04,A -85,B 0,C 180,E1 -3078.43,E2 -3078.43} C_VEL
LIN {X 0,Y 552.657,Z 344.937,A -85,B 0,C 180,E1 -3078.951,E2 -3078.951} C_VEL
LIN {X 0,Y 552.843,Z 330.799,A -85,B 0,C 180,E1 -3081.242,E2 -3081.242} C_VEL
LIN {X 0,Y 552.134,Z 325.338,A -85,B 0,C 180,E1 -3082.17,E2 -3082.17} C_VEL
LIN {X 0,Y 552.143,Z 325.329,A -85,B 0,C 180,E1 -3085.346,E2 -3085.346} C_VEL
LIN {X 0,Y 552.095,Z 325.342,A -85,B 0,C 180,E1 -3088.099,E2 -3088.099} C_VEL
LIN {X 0,Y 552.106,Z 325.334,A -85,B 0,C 180,E1 -3090.609,E2 -3090.609} C_VEL
LIN {X 0,Y 552.12,Z 325.331,A -85,B 0,C 180,E1 -3093.186,E2 -3093.186} C_VEL
LIN {X 0,Y 552.079,Z 325.343,A -85,B 0,C 180,E1 -3095.844,E2 -3095.844} C_VEL
LIN {X 0,Y 552.119,Z 325.331,A -85,B 0,C 180,E1 -3098.589,E2 -3098.589} C_VEL
LIN {X 0,Y 552.115,Z 325.335,A -85,B 0,C 180,E1 -3101.447,E2 -3101.447} C_VEL
LIN {X 0,Y 552.093,Z 325.335,A -85,B 0,C 180,E1 -3104.531,E2 -3104.531} C_VEL
LIN {X 0,Y 552.114,Z 325.34,A -85,B 0,C 180,E1 -3107.587,E2 -3107.587} C_VEL
LIN {X 0,Y 552.13,Z 325.33,A -85,B 0,C 180,E1 -3110.472,E2 -3110.472} C_VEL
LIN {X 0,Y 552.101,Z 325.34,A -85,B 0,C 180,E1 -3113.318,E2 -3113.318} C_VEL
LIN {X 0,Y 552.094,Z 325.337,A -85,B 0,C 180,E1 -3115.936,E2 -3115.936} C_VEL
LIN {X 0,Y 552.084,Z 325.336,A -85,B 0,C 180,E1 -3118.537,E2 -3118.537} C_VEL
LIN {X 0,Y 552.081,Z 325.343,A -85,B 0,C 180,E1 -3121.447,E2 -3121.447} C_VEL
LIN {X 0,Y 552.046,Z 325.342,A -85,B 0,C 180,E1 -3124.351,E2 -3124.351} C_VEL
LIN {X 0,Y 552.109,Z 325.432,A -85,B 0,C 180,E1 -3126.956,E2 -3126.956} C_VEL
LIN {X 0,Y 553.197,Z 332.065,A -85,B 0,C 180,E1 -3128.036,E2 -3128.036} C_VEL
LIN {X 0,Y 552.847,Z 349.506,A -85,B 0,C 180,E1 -3130.699,E2 -3130.699} C_VEL
LIN {X 0,Y 552.663,Z 362.32,A -85,B 0,C 180,E1 -3132.631,E2 -3132.631} C_VEL
LIN {X 0,Y 554.259,Z 371.91,A -85,B 0,C 180,E1 -3132.816,E2 -3132.816} C_VEL
LIN {X 0,Y 553.736,Z 498.208,A -85,B 0,C 180,E1 -3134.494,E2 -3134.494} C_VEL
LIN {X 0,Y 553.627,Z 509.573,A -85,B 0,C 180,E1 -3134.739,E2 -3134.739} C_VEL
LIN {X 0,Y 553.542,Z 519.541,A -85,B 0,C 180,E1 -3135.035,E2 -3135.035} C_VEL
LIN {X 0,Y 553.355,Z 529.849,A -85,B 0,C 180,E1 -3135.425,E2 -3135.425} C_VEL
LIN {X 0,Y 553.147,Z 540.661,A -85,B 0,C 180,E1 -3135.936,E2 -3135.936} C_VEL
LIN {X 0,Y 552.928,Z 550.416,A -85,B 0,C 180,E1 -3136.493,E2 -3136.493} C_VEL
LIN {X 0,Y 552.743,Z 559.997,A -85,B 0,C 180,E1 -3137.143,E2 -3137.143} C_VEL
LIN {X 0,Y 552.542,Z 569.286,A -85,B 0,C 180,E1 -3137.884,E2 -3137.884} C_VEL
LIN {X 0,Y 552.399,Z 578.53,A -85,B 0,C 180,E1 -3138.752,E2 -3138.752} C_VEL
LIN {X 0,Y 552.236,Z 585.858,A -85,B 0,C 180,E1 -3139.551,E2 -3139.551} C_VEL
LIN {X 0,Y 552.073,Z 593.172,A -85,B 0,C 180,E1 -3140.473,E2 -3140.473} C_VEL
LIN {X 0,Y 551.963,Z 599.456,A -85,B 0,C 180,E1 -3141.395,E2 -3141.395} C_VEL
LIN {X 0,Y 551.903,Z 604.874,A -85,B 0,C 180,E1 -3142.315,E2 -3142.315} C_VEL
LIN {X 0,Y 551.824,Z 610.307,A -85,B 0,C 180,E1 -3143.417,E2 -3143.417} C_VEL
LIN {X 0,Y 551.792,Z 614.75,A -85,B 0,C 180,E1 -3144.517,E2 -3144.517} C_VEL
LIN {X 0,Y 551.76,Z 618.304,A -85,B 0,C 180,E1 -3145.616,E2 -3145.616} C_VEL
LIN {X 0,Y 551.741,Z 620.213,A -85,B 0,C 180,E1 -3146.347,E2 -3146.347} C_VEL
LIN {X 0,Y 551.656,Z 622.943,A -85,B 0,C 180,E1 -3147.809,E2 -3147.809} C_VEL
LIN {X 0,Y 551.637,Z 624.258,A -85,B 0,C 180,E1 -3149.269,E2 -3149.269} C_VEL
LIN {X 0,Y 551.64,Z 624.496,A -85,B 0,C 180,E1 -3149.999,E2 -3149.999} C_VEL
LIN {X 0,Y 551.64,Z 623.851,A -85,B 0,C 180,E1 -3151.459,E2 -3151.459} C_VEL
LIN {X 0,Y 551.718,Z 621.868,A -85,B 0,C 180,E1 -3152.92,E2 -3152.92} C_VEL
LIN {X 0,Y 551.741,Z 620.437,A -85,B 0,C 180,E1 -3153.65,E2 -3153.65} C_VEL
LIN {X 0,Y 551.716,Z 616.321,A -85,B 0,C 180,E1 -3155.115,E2 -3155.115} C_VEL
LIN {X 0,Y 551.819,Z 613.773,A -85,B 0,C 180,E1 -3155.847,E2 -3155.847} C_VEL
LIN {X 0,Y 551.829,Z 607.25,A -85,B 0,C 180,E1 -3157.316,E2 -3157.316} C_VEL
LIN {X 0,Y 551.96,Z 601.153,A -85,B 0,C 180,E1 -3158.419,E2 -3158.419} C_VEL
LIN {X 0,Y 552.061,Z 595.167,A -85,B 0,C 180,E1 -3159.34,E2 -3159.34} C_VEL
LIN {X 0,Y 552.173,Z 588.187,A -85,B 0,C 180,E1 -3160.263,E2 -3160.263} C_VEL
LIN {X 0,Y 552.355,Z 579.454,A -85,B 0,C 180,E1 -3161.244,E2 -3161.244} C_VEL
LIN {X 0,Y 552.51,Z 570.331,A -85,B 0,C 180,E1 -3162.114,E2 -3162.114} C_VEL
LIN {X 0,Y 552.703,Z 561.218,A -85,B 0,C 180,E1 -3162.856,E2 -3162.856} C_VEL
LIN {X 0,Y 552.916,Z 551.855,A -85,B 0,C 180,E1 -3163.506,E2 -3163.506} C_VEL
LIN {X 0,Y 553.095,Z 542.382,A -85,B 0,C 180,E1 -3164.063,E2 -3164.063} C_VEL
LIN {X 0,Y 553.28,Z 531.953,A -85,B 0,C 180,E1 -3164.575,E2 -3164.575} C_VEL
LIN {X 0,Y 553.525,Z 521.206,A -85,B 0,C 180,E1 -3164.998,E2 -3164.998} C_VEL
LIN {X 0,Y 553.62,Z 510.119,A -85,B 0,C 180,E1 -3165.338,E2 -3165.338} C_VEL
LIN {X 0,Y 553.73,Z 499.447,A -85,B 0,C 180,E1 -3165.575,E2 -3165.575} C_VEL
LIN {X 0,Y 553.922,Z 465.711,A -85,B 0,C 180,E1 -3166.041,E2 -3166.041} C_VEL
LIN {X 0,Y 554.099,Z 370.078,A -85,B 0,C 180,E1 -3167.303,E2 -3167.303} C_VEL
LIN {X 0,Y 552.659,Z 362.311,A -85,B 0,C 180,E1 -3167.461,E2 -3167.461} C_VEL
LIN {X 0,Y 553.044,Z 341.248,A -85,B 0,C 180,E1 -3170.648,E2 -3170.648} C_VEL
LIN {X 0,Y 553.173,Z 331.668,A -85,B 0,C 180,E1 -3172.119,E2 -3172.119} C_VEL
LIN {X 0,Y 552.103,Z 325.342,A -85,B 0,C 180,E1 -3173.166,E2 -3173.166} C_VEL
LIN {X 0,Y 552.072,Z 325.34,A -85,B 0,C 180,E1 -3175.646,E2 -3175.646} C_VEL
LIN {X 0,Y 552.073,Z 325.341,A -85,B 0,C 180,E1 -3178.552,E2 -3178.552} C_VEL
LIN {X 0,Y 552.085,Z 325.339,A -85,B 0,C 180,E1 -3181.471,E2 -3181.471} C_VEL
LIN {X 0,Y 552.116,Z 325.333,A -85,B 0,C 180,E1 -3184.167,E2 -3184.167} C_VEL
LIN {X 0,Y 552.089,Z 325.342,A -85,B 0,C 180,E1 -3186.747,E2 -3186.747} C_VEL
LIN {X 0,Y 552.115,Z 325.333,A -85,B 0,C 180,E1 -3189.526,E2 -3189.526} C_VEL
LIN {X 0,Y 552.073,Z 325.339,A -85,B 0,C 180,E1 -3192.429,E2 -3192.429} C_VEL
LIN {X 0,Y 552.068,Z 325.338,A -85,B 0,C 180,E1 -3195.559,E2 -3195.559} C_VEL
LIN {X 0,Y 552.062,Z 325.342,A -85,B 0,C 180,E1 -3198.548,E2 -3198.548} C_VEL
LIN {X 0,Y 552.098,Z 325.332,A -85,B 0,C 180,E1 -3201.409,E2 -3201.409} C_VEL
LIN {X 0,Y 552.057,Z 325.339,A -85,B 0,C 180,E1 -3204.154,E2 -3204.154} C_VEL
LIN {X 0,Y 552.093,Z 325.335,A -85,B 0,C 180,E1 -3207.154,E2 -3207.154} C_VEL
LIN {X 0,Y 552.075,Z 325.336,A -85,B 0,C 180,E1 -3209.954,E2 -3209.954} C_VEL
LIN {X 0,Y 552.078,Z 325.337,A -85,B 0,C 180,E1 -3213.009,E2 -3213.009} C_VEL
LIN {X 0,Y 552.062,Z 325.337,A -85,B 0,C 180,E1 -3215.96,E2 -3215.96} C_VEL
LIN {X 0,Y 552.099,Z 325.333,A -85,B 0,C 180,E1 -3219.119,E2 -3219.119} C_VEL
LIN {X 0,Y 552.067,Z 325.334,A -85,B 0,C 180,E1 -3221.442,E2 -3221.442} C_VEL
LIN {X 0,Y 552.073,Z 325.336,A -85,B 0,C 180,E1 -3223.736,E2 -3223.736} C_VEL
LIN {X 0,Y 552.088,Z 325.335,A -85,B 0,C 180,E1 -3226.003,E2 -3226.003} C_VEL
LIN {X 0,Y 552.134,Z 325.332,A -85,B 0,C 180,E1 -3228.993,E2 -3228.993} C_VEL
LIN {X 0,Y 552.125,Z 325.33,A -85,B 0,C 180,E1 -3231.951,E2 -3231.951} C_VEL
LIN {X 0,Y 552.193,Z 325.325,A -85,B 0,C 180,E1 -3234.889,E2 -3234.889} C_VEL
LIN {X 0,Y 552.189,Z 325.322,A -85,B 0,C 180,E1 -3237.812,E2 -3237.812} C_VEL
LIN {X 0,Y 552.225,Z 325.324,A -85,B 0,C 180,E1 -3240.729,E2 -3240.729} C_VEL
LIN {X 0,Y 552.174,Z 325.327,A -85,B 0,C 180,E1 -3242.918,E2 -3242.918} C_VEL
LIN {X 0,Y 552.157,Z 325.326,A -85,B 0,C 180,E1 -3245.844,E2 -3245.844} C_VEL
LIN {X 0,Y 552.111,Z 325.336,A -85,B 0,C 180,E1 -3248.786,E2 -3248.786} C_VEL
LIN {X 0,Y 552.093,Z 325.334,A -85,B 0,C 180,E1 -3251.752,E2 -3251.752} C_VEL
LIN {X 0,Y 552.119,Z 325.335,A -85,B 0,C 180,E1 -3254.749,E2 -3254.749} C_VEL
LIN {X 0,Y 552.069,Z 325.337,A -85,B 0,C 180,E1 -3257.79,E2 -3257.79} C_VEL
LIN {X 0,Y 552.109,Z 325.336,A -85,B 0,C 180,E1 -3260.102,E2 -3260.102} C_VEL
LIN {X 0,Y 552.07,Z 325.341,A -85,B 0,C 180,E1 -3262.452,E2 -3262.452} C_VEL
LIN {X 0,Y 552.063,Z 325.337,A -85,B 0,C 180,E1 -3265.334,E2 -3265.334} C_VEL
LIN {X 0,Y 552.061,Z 325.342,A -85,B 0,C 180,E1 -3268.101,E2 -3268.101} C_VEL
LIN {X 0,Y 552.072,Z 325.342,A -85,B 0,C 180,E1 -3270.611,E2 -3270.611} C_VEL
LIN {X 0,Y 552.089,Z 325.333,A -85,B 0,C 180,E1 -3273.188,E2 -3273.188} C_VEL
LIN {X 0,Y 552.053,Z 325.341,A -85,B 0,C 180,E1 -3275.846,E2 -3275.846} C_VEL
LIN {X 0,Y 552.096,Z 325.338,A -85,B 0,C 180,E1 -3278.591,E2 -3278.591} C_VEL
LIN {X 0,Y 552.04,Z 325.34,A -85,B 0,C 180,E1 -3281.453,E2 -3281.453} C_VEL
LIN {X 0,Y 552.059,Z 325.343,A -85,B 0,C 180,E1 -3284.53,E2 -3284.53} C_VEL
LIN {X 0,Y 552.068,Z 325.339,A -85,B 0,C 180,E1 -3287.592,E2 -3287.592} C_VEL
LIN {X 0,Y 552.077,Z 325.337,A -85,B 0,C 180,E1 -3290.945,E2 -3290.945} C_VEL
LIN {X 0,Y 552.041,Z 325.341,A -85,B 0,C 180,E1 -3293.326,E2 -3293.326} C_VEL
LIN {X 0,Y 552.086,Z 325.341,A -85,B 0,C 180,E1 -3295.938,E2 -3295.938} C_VEL
LIN {X 0,Y 552.096,Z 325.337,A -85,B 0,C 180,E1 -3298.541,E2 -3298.541} C_VEL
LIN {X 0,Y 552.063,Z 325.338,A -85,B 0,C 180,E1 -3301.45,E2 -3301.45} C_VEL
LIN {X 0,Y 552.061,Z 325.346,A -85,B 0,C 180,E1 -3304.354,E2 -3304.354} C_VEL
LIN {X 0,Y 552.131,Z 325.494,A -85,B 0,C 180,E1 -3305.84,E2 -3305.84} C_VEL
LIN {X 0,Y 553.318,Z 331.736,A -85,B 0,C 180,E1 -3306.814,E2 -3306.814} C_VEL
LIN {X 0,Y 553.181,Z 345.219,A -85,B 0,C 180,E1 -3308.773,E2 -3308.773} C_VEL
LIN {X 0,Y 552.797,Z 364.084,A -85,B 0,C 180,E1 -3311.469,E2 -3311.469} C_VEL
LIN {X 0,Y 552.729,Z 371.97,A -85,B 0,C 180,E1 -3312.588,E2 -3312.588} C_VEL
LIN {X 0,Y 554.205,Z 380.614,A -85,B 0,C 180,E1 -3312.752,E2 -3312.752} C_VEL
LIN {X 0,Y 553.778,Z 508.711,A -85,B 0,C 180,E1 -3314.45,E2 -3314.45} C_VEL
LIN {X 0,Y 553.603,Z 523.289,A -85,B 0,C 180,E1 -3314.788,E2 -3314.788} C_VEL
LIN {X 0,Y 553.371,Z 537.727,A -85,B 0,C 180,E1 -3315.287,E2 -3315.287} C_VEL
LIN {X 0,Y 553.16,Z 551.664,A -85,B 0,C 180,E1 -3315.938,E2 -3315.938} C_VEL
LIN {X 0,Y 552.878,Z 564.122,A -85,B 0,C 180,E1 -3316.681,E2 -3316.681} C_VEL
LIN {X 0,Y 552.629,Z 576.662,A -85,B 0,C 180,E1 -3317.609,E2 -3317.609} C_VEL
LIN {X 0,Y 552.445,Z 587.306,A -85,B 0,C 180,E1 -3318.574,E2 -3318.574} C_VEL
LIN {X 0,Y 552.178,Z 597.862,A -85,B 0,C 180,E1 -3319.737,E2 -3319.737} C_VEL
LIN {X 0,Y 552.031,Z 606.183,A -85,B 0,C 180,E1 -3320.844,E2 -3320.844} C_VEL
LIN {X 0,Y 551.912,Z 614.134,A -85,B 0,C 180,E1 -3322.133,E2 -3322.133} C_VEL
LIN {X 0,Y 551.82,Z 620.532,A -85,B 0,C 180,E1 -3323.419,E2 -3323.419} C_VEL
LIN {X 0,Y 551.791,Z 624.964,A -85,B 0,C 180,E1 -3324.52,E2 -3324.52} C_VEL
LIN {X 0,Y 551.759,Z 628.45,A -85,B 0,C 180,E1 -3325.618,E2 -3325.618} C_VEL
LIN {X 0,Y 551.72,Z 631.837,A -85,B 0,C 180,E1 -3327.08,E2 -3327.08} C_VEL
LIN {X 0,Y 551.64,Z 633.836,A -85,B 0,C 180,E1 -3328.541,E2 -3328.541} C_VEL
LIN {X 0,Y 551.639,Z 634.5,A -85,B 0,C 180,E1 -3330.001,E2 -3330.001} C_VEL
LIN {X 0,Y 551.64,Z 633.833,A -85,B 0,C 180,E1 -3331.461,E2 -3331.461} C_VEL
LIN {X 0,Y 551.72,Z 631.83,A -85,B 0,C 180,E1 -3332.922,E2 -3332.922} C_VEL
LIN {X 0,Y 551.76,Z 628.441,A -85,B 0,C 180,E1 -3334.384,E2 -3334.384} C_VEL
LIN {X 0,Y 551.818,Z 623.565,A -85,B 0,C 180,E1 -3335.849,E2 -3335.849} C_VEL
LIN {X 0,Y 551.834,Z 617.049,A -85,B 0,C 180,E1 -3337.318,E2 -3337.318} C_VEL
LIN {X 0,Y 551.963,Z 609.796,A -85,B 0,C 180,E1 -3338.605,E2 -3338.605} C_VEL
LIN {X 0,Y 552.117,Z 600.814,A -85,B 0,C 180,E1 -3339.896,E2 -3339.896} C_VEL
LIN {X 0,Y 552.348,Z 591.383,A -85,B 0,C 180,E1 -3341.004,E2 -3341.004} C_VEL
LIN {X 0,Y 552.54,Z 580.943,A -85,B 0,C 180,E1 -3342.023,E2 -3342.023} C_VEL
LIN {X 0,Y 552.762,Z 569.415,A -85,B 0,C 180,E1 -3342.95,E2 -3342.95} C_VEL
LIN {X 0,Y 553.018,Z 556.62,A -85,B 0,C 180,E1 -3343.786,E2 -3343.786} C_VEL
LIN {X 0,Y 553.269,Z 544.132,A -85,B 0,C 180,E1 -3344.436,E2 -3344.436} C_VEL
LIN {X 0,Y 553.503,Z 530.931,A -85,B 0,C 180,E1 -3344.969,E2 -3344.969} C_VEL
LIN {X 0,Y 553.664,Z 516.848,A -85,B 0,C 180,E1 -3345.381,E2 -3345.381} C_VEL
LIN {X 0,Y 553.787,Z 502.535,A -85,B 0,C 180,E1 -3345.646,E2 -3345.646} C_VEL
LIN {X 0,Y 554.143,Z 379.693,A -85,B 0,C 180,E1 -3347.262,E2 -3347.262} C_VEL
LIN {X 0,Y 552.704,Z 371.804,A -85,B 0,C 180,E1 -3347.436,E2 -3347.436} C_VEL
LIN {X 0,Y 553.135,Z 349.248,A -85,B 0,C 180,E1 -3350.646,E2 -3350.646} C_VEL
LIN {X 0,Y 553.434,Z 333.072,A -85,B 0,C 180,E1 -3352.986,E2 -3352.986} C_VEL
LIN {X 0,Y 552.113,Z 325.34,A -85,B 0,C 180,E1 -3354.188,E2 -3354.188} C_VEL
LIN {X 0,Y 552.066,Z 325.344,A -85,B 0,C 180,E1 -3357.278,E2 -3357.278} C_VEL
LIN {X 0,Y 552.092,Z 325.338,A -85,B 0,C 180,E1 -3360.046,E2 -3360.046} C_VEL
LIN {X 0,Y 552.114,Z 325.334,A -85,B 0,C 180,E1 -3362.846,E2 -3362.846} C_VEL
LIN {X 0,Y 552.074,Z 325.343,A -85,B 0,C 180,E1 -3365.439,E2 -3365.439} C_VEL
LIN {X 0,Y 552.098,Z 325.334,A -85,B 0,C 180,E1 -3367.886,E2 -3367.886} C_VEL
LIN {X 0,Y 552.114,Z 325.333,A -85,B 0,C 180,E1 -3370.482,E2 -3370.482} C_VEL
LIN {X 0,Y 552.111,Z 325.335,A -85,B 0,C 180,E1 -3373.424,E2 -3373.424} C_VEL
LIN {X 0,Y 552.113,Z 325.339,A -85,B 0,C 180,E1 -3376.577,E2 -3376.577} C_VEL
LIN {X 0,Y 552.113,Z 325.332,A -85,B 0,C 180,E1 -3379.519,E2 -3379.519} C_VEL
LIN {X 0,Y 552.093,Z 325.341,A -85,B 0,C 180,E1 -3382.336,E2 -3382.336} C_VEL
LIN {X 0,Y 552.086,Z 325.337,A -85,B 0,C 180,E1 -3385.051,E2 -3385.051} C_VEL
LIN {X 0,Y 552.119,Z 325.334,A -85,B 0,C 180,E1 -3387.682,E2 -3387.682} C_VEL
LIN {X 0,Y 552.113,Z 325.341,A -85,B 0,C 180,E1 -3390.235,E2 -3390.235} C_VEL
LIN {X 0,Y 552.082,Z 325.339,A -85,B 0,C 180,E1 -3393.013,E2 -3393.013} C_VEL
LIN {X 0,Y 552.088,Z 325.344,A -85,B 0,C 180,E1 -3395.961,E2 -3395.961} C_VEL
LIN {X 0,Y 552.113,Z 325.349,A -85,B 0,C 180,E1 -3397.998,E2 -3397.998} C_VEL
LIN {X 0,Y 552.85,Z 331.19,A -85,B 0,C 180,E1 -3398.954,E2 -3398.954} C_VEL
LIN {X 0,Y 552.612,Z 349.233,A -85,B 0,C 180,E1 -3401.845,E2 -3401.845} C_VEL
LIN {X 0,Y 552.478,Z 359.946,A -85,B 0,C 180,E1 -3403.558,E2 -3403.558} C_VEL
LIN {X 0,Y 552.339,Z 373.167,A -85,B 0,C 180,E1 -3405.686,E2 -3405.686} C_VEL
LIN {X 0,Y 553.428,Z 380.813,A -85,B 0,C 180,E1 -3405.815,E2 -3405.815} C_VEL
LIN {X 0,Y 553.106,Z 480.406,A -85,B 0,C 180,E1 -3407.129,E2 -3407.129} C_VEL
LIN {X 0,Y 552.994,Z 493.765,A -85,B 0,C 180,E1 -3407.453,E2 -3407.453} C_VEL
LIN {X 0,Y 552.857,Z 505.893,A -85,B 0,C 180,E1 -3407.893,E2 -3407.893} C_VEL
LIN {X 0,Y 552.675,Z 518.527,A -85,B 0,C 180,E1 -3408.513,E2 -3408.513} C_VEL
LIN {X 0,Y 552.474,Z 530.39,A -85,B 0,C 180,E1 -3409.278,E2 -3409.278} C_VEL
LIN {X 0,Y 552.276,Z 540.584,A -85,B 0,C 180,E1 -3410.108,E2 -3410.108} C_VEL
LIN {X 0,Y 552.123,Z 549.889,A -85,B 0,C 180,E1 -3411.029,E2 -3411.029} C_VEL
LIN {X 0,Y 551.985,Z 557.468,A -85,B 0,C 180,E1 -3411.949,E2 -3411.949} C_VEL
LIN {X 0,Y 551.873,Z 565.181,A -85,B 0,C 180,E1 -3413.088,E2 -3413.088} C_VEL
LIN {X 0,Y 551.868,Z 570.944,A -85,B 0,C 180,E1 -3414.153,E2 -3414.153} C_VEL
LIN {X 0,Y 551.739,Z 575.712,A -85,B 0,C 180,E1 -3415.251,E2 -3415.251} C_VEL
LIN {X 0,Y 551.751,Z 579.304,A -85,B 0,C 180,E1 -3416.349,E2 -3416.349} C_VEL
LIN {X 0,Y 551.724,Z 581.167,A -85,B 0,C 180,E1 -3417.079,E2 -3417.079} C_VEL
LIN {X 0,Y 551.645,Z 583.64,A -85,B 0,C 180,E1 -3418.54,E2 -3418.54} C_VEL
LIN {X 0,Y 551.642,Z 584.273,A -85,B 0,C 180,E1 -3419.27,E2 -3419.27} C_VEL
LIN {X 0,Y 551.641,Z 584.496,A -85,B 0,C 180,E1 -3420,E2 -3420} C_VEL
LIN {X 0,Y 551.642,Z 584.31,A -85,B 0,C 180,E1 -3420.73,E2 -3420.73} C_VEL
LIN {X 0,Y 551.645,Z 583.724,A -85,B 0,C 180,E1 -3421.46,E2 -3421.46} C_VEL
LIN {X 0,Y 551.724,Z 581.366,A -85,B 0,C 180,E1 -3422.921,E2 -3422.921} C_VEL
LIN {X 0,Y 551.764,Z 578.516,A -85,B 0,C 180,E1 -3424.017,E2 -3424.017} C_VEL
LIN {X 0,Y 551.724,Z 574.616,A -85,B 0,C 180,E1 -3425.116,E2 -3425.116} C_VEL
LIN {X 0,Y 551.811,Z 568.891,A -85,B 0,C 180,E1 -3426.348,E2 -3426.348} C_VEL
LIN {X 0,Y 551.926,Z 562.01,A -85,B 0,C 180,E1 -3427.5,E2 -3427.5} C_VEL
LIN {X 0,Y 552.06,Z 553.865,A -85,B 0,C 180,E1 -3428.603,E2 -3428.603} C_VEL
LIN {X 0,Y 552.196,Z 545.424,A -85,B 0,C 180,E1 -3429.524,E2 -3429.524} C_VEL
LIN {X 0,Y 552.396,Z 535.129,A -85,B 0,C 180,E1 -3430.446,E2 -3430.446} C_VEL
LIN {X 0,Y 552.581,Z 524.52,A -85,B 0,C 180,E1 -3431.213,E2 -3431.213} C_VEL
LIN {X 0,Y 552.727,Z 513.772,A -85,B 0,C 180,E1 -3431.831,E2 -3431.831} C_VEL
LIN {X 0,Y 552.907,Z 501.224,A -85,B 0,C 180,E1 -3432.386,E2 -3432.386} C_VEL
LIN {X 0,Y 553.053,Z 488.74,A -85,B 0,C 180,E1 -3432.779,E2 -3432.779} C_VEL
LIN {X 0,Y 553.16,Z 476.063,A -85,B 0,C 180,E1 -3433.033,E2 -3433.033} C_VEL
LIN {X 0,Y 553.308,Z 379.04,A -85,B 0,C 180,E1 -3434.302,E2 -3434.302} C_VEL
LIN {X 0,Y 552.317,Z 372.957,A -85,B 0,C 180,E1 -3434.408,E2 -3434.408} C_VEL
LIN {X 0,Y 552.593,Z 354.13,A -85,B 0,C 180,E1 -3437.47,E2 -3437.47} C_VEL
LIN {X 0,Y 552.657,Z 344.937,A -85,B 0,C 180,E1 -3438.951,E2 -3438.951} C_VEL
LIN {X 0,Y 552.103,Z 341.871,A -85,B 0,C 180,E1 -3439.47,E2 -3439.47} C_VEL
LIN {X 0,Y 546.181,Z 331.472,A -85,B 0,C 180,E1 -3441.38,E2 -3441.38} C_VEL
LIN {X 0,Y 545.678,Z 329.41,A -85,B 0,C 180,E1 -3441.734,E2 -3441.734} C_VEL
LIN {X 0,Y 545.084,Z 326.216,A -85,B 0,C 180,E1 -3442.306,E2 -3442.306} C_VEL
LIN {X 0,Y 545.091,Z 326.208,A -85,B 0,C 180,E1 -3445.507,E2 -3445.507} C_VEL
LIN {X 0,Y 545.088,Z 326.211,A -85,B 0,C 180,E1 -3448.493,E2 -3448.493} C_VEL
LIN {X 0,Y 545.071,Z 326.208,A -85,B 0,C 180,E1 -3451.048,E2 -3451.048} C_VEL
LIN {X 0,Y 545.07,Z 326.213,A -85,B 0,C 180,E1 -3453.672,E2 -3453.672} C_VEL
LIN {X 0,Y 545.07,Z 326.209,A -85,B 0,C 180,E1 -3456.925,E2 -3456.925} C_VEL
LIN {X 0,Y 545.07,Z 326.214,A -85,B 0,C 180,E1 -3460.142,E2 -3460.142} C_VEL
LIN {X 0,Y 545.05,Z 326.213,A -85,B 0,C 180,E1 -3463.11,E2 -3463.11} C_VEL
LIN {X 0,Y 545.05,Z 326.214,A -85,B 0,C 180,E1 -3466.226,E2 -3466.226} C_VEL
LIN {X 0,Y 545.033,Z 326.214,A -85,B 0,C 180,E1 -3468.88,E2 -3468.88} C_VEL
LIN {X 0,Y 545.048,Z 326.218,A -85,B 0,C 180,E1 -3471.761,E2 -3471.761} C_VEL
LIN {X 0,Y 545.029,Z 326.214,A -85,B 0,C 180,E1 -3474.53,E2 -3474.53} C_VEL
LIN {X 0,Y 545.055,Z 326.218,A -85,B 0,C 180,E1 -3477.21,E2 -3477.21} C_VEL
LIN {X 0,Y 545.028,Z 326.218,A -85,B 0,C 180,E1 -3479.807,E2 -3479.807} C_VEL
LIN {X 0,Y 545.003,Z 326.218,A -85,B 0,C 180,E1 -3482.339,E2 -3482.339} C_VEL
LIN {X 0,Y 545.02,Z 326.222,A -85,B 0,C 180,E1 -3484.815,E2 -3484.815} C_VEL
LIN {X 0,Y 545.061,Z 326.289,A -85,B 0,C 180,E1 -3486.766,E2 -3486.766} C_VEL
LIN {X 0,Y 546.264,Z 332.931,A -85,B 0,C 180,E1 -3487.869,E2 -3487.869} C_VEL
LIN {X 0,Y 546.014,Z 348.454,A -85,B 0,C 180,E1 -3490.276,E2 -3490.276} C_VEL
LIN {X 0,Y 545.72,Z 362.342,A -85,B 0,C 180,E1 -3492.396,E2 -3492.396} C_VEL
LIN {X 0,Y 547.472,Z 372.302,A -85,B 0,C 180,E1 -3492.6,E2 -3492.6} C_VEL
LIN {X 0,Y 546.897,Z 498.256,A -85,B 0,C 180,E1 -3494.295,E2 -3494.295} C_VEL
LIN {X 0,Y 546.785,Z 509.633,A -85,B 0,C 180,E1 -3494.544,E2 -3494.544} C_VEL
LIN {X 0,Y 546.702,Z 518.398,A -85,B 0,C 180,E1 -3494.803,E2 -3494.803} C_VEL
LIN {X 0,Y 546.45,Z 529.839,A -85,B 0,C 180,E1 -3495.237,E2 -3495.237} C_VEL
LIN {X 0,Y 546.254,Z 540.659,A -85,B 0,C 180,E1 -3495.755,E2 -3495.755} C_VEL
LIN {X 0,Y 545.989,Z 550.408,A -85,B 0,C 180,E1 -3496.318,E2 -3496.318} C_VEL
LIN {X 0,Y 545.791,Z 559.99,A -85,B 0,C 180,E1 -3496.976,E2 -3496.976} C_VEL
LIN {X 0,Y 545.567,Z 569.283,A -85,B 0,C 180,E1 -3497.727,E2 -3497.727} C_VEL
LIN {X 0,Y 545.397,Z 577.386,A -85,B 0,C 180,E1 -3498.488,E2 -3498.488} C_VEL
LIN {X 0,Y 545.224,Z 585.852,A -85,B 0,C 180,E1 -3499.415,E2 -3499.415} C_VEL
LIN {X 0,Y 545.026,Z 593.167,A -85,B 0,C 180,E1 -3500.349,E2 -3500.349} C_VEL
LIN {X 0,Y 544.911,Z 599.453,A -85,B 0,C 180,E1 -3501.282,E2 -3501.282} C_VEL
LIN {X 0,Y 544.826,Z 604.868,A -85,B 0,C 180,E1 -3502.215,E2 -3502.215} C_VEL
LIN {X 0,Y 544.736,Z 610.714,A -85,B 0,C 180,E1 -3503.429,E2 -3503.429} C_VEL
LIN {X 0,Y 544.724,Z 614.745,A -85,B 0,C 180,E1 -3504.446,E2 -3504.446} C_VEL
LIN {X 0,Y 544.655,Z 618.298,A -85,B 0,C 180,E1 -3505.559,E2 -3505.559} C_VEL
LIN {X 0,Y 544.658,Z 620.216,A -85,B 0,C 180,E1 -3506.3,E2 -3506.3} C_VEL
LIN {X 0,Y 544.57,Z 622.939,A -85,B 0,C 180,E1 -3507.78,E2 -3507.78} C_VEL
LIN {X 0,Y 544.537,Z 624.251,A -85,B 0,C 180,E1 -3509.259,E2 -3509.259} C_VEL
LIN {X 0,Y 544.54,Z 624.496,A -85,B 0,C 180,E1 -3509.999,E2 -3509.999} C_VEL
LIN {X 0,Y 544.542,Z 623.847,A -85,B 0,C 180,E1 -3511.478,E2 -3511.478} C_VEL
LIN {X 0,Y 544.645,Z 621.86,A -85,B 0,C 180,E1 -3512.958,E2 -3512.958} C_VEL
LIN {X 0,Y 544.658,Z 620.436,A -85,B 0,C 180,E1 -3513.698,E2 -3513.698} C_VEL
LIN {X 0,Y 544.645,Z 616.313,A -85,B 0,C 180,E1 -3515.181,E2 -3515.181} C_VEL
LIN {X 0,Y 544.691,Z 612.199,A -85,B 0,C 180,E1 -3516.309,E2 -3516.309} C_VEL
LIN {X 0,Y 544.78,Z 607.238,A -85,B 0,C 180,E1 -3517.411,E2 -3517.411} C_VEL
LIN {X 0,Y 544.894,Z 601.142,A -85,B 0,C 180,E1 -3518.529,E2 -3518.529} C_VEL
LIN {X 0,Y 545.016,Z 595.153,A -85,B 0,C 180,E1 -3519.462,E2 -3519.462} C_VEL
LIN {X 0,Y 545.15,Z 588.171,A -85,B 0,C 180,E1 -3520.397,E2 -3520.397} C_VEL
LIN {X 0,Y 545.334,Z 580.106,A -85,B 0,C 180,E1 -3521.321,E2 -3521.321} C_VEL
LIN {X 0,Y 545.517,Z 571.372,A -85,B 0,C 180,E1 -3522.177,E2 -3522.177} C_VEL
LIN {X 0,Y 545.726,Z 562.433,A -85,B 0,C 180,E1 -3522.929,E2 -3522.929} C_VEL
LIN {X 0,Y 545.938,Z 553.29,A -85,B 0,C 180,E1 -3523.587,E2 -3523.587} C_VEL
LIN {X 0,Y 546.202,Z 542.358,A -85,B 0,C 180,E1 -3524.244,E2 -3524.244} C_VEL
LIN {X 0,Y 546.39,Z 531.916,A -85,B 0,C 180,E1 -3524.763,E2 -3524.763} C_VEL
LIN {X 0,Y 546.641,Z 521.161,A -85,B 0,C 180,E1 -3525.191,E2 -3525.191} C_VEL
LIN {X 0,Y 546.77,Z 510.307,A -85,B 0,C 180,E1 -3525.529,E2 -3525.529} C_VEL
LIN {X 0,Y 546.888,Z 499.424,A -85,B 0,C 180,E1 -3525.775,E2 -3525.775} C_VEL
LIN {X 0,Y 547.117,Z 465.691,A -85,B 0,C 180,E1 -3526.246,E2 -3526.246} C_VEL
LIN {X 0,Y 547.311,Z 371.069,A -85,B 0,C 180,E1 -3527.512,E2 -3527.512} C_VEL
LIN {X 0,Y 545.706,Z 362.247,A -85,B 0,C 180,E1 -3527.709,E2 -3527.709} C_VEL
LIN {X 0,Y 546.11,Z 342.573,A -85,B 0,C 180,E1 -3530.725,E2 -3530.725} C_VEL
LIN {X 0,Y 546.155,Z 332.092,A -85,B 0,C 180,E1 -3532.359,E2 -3532.359} C_VEL
LIN {X 0,Y 545.063,Z 326.218,A -85,B 0,C 180,E1 -3533.357,E2 -3533.357} C_VEL
LIN {X 0,Y 545.033,Z 326.216,A -85,B 0,C 180,E1 -3536.001,E2 -3536.001} C_VEL
LIN {X 0,Y 545.038,Z 326.22,A -85,B 0,C 180,E1 -3538.738,E2 -3538.738} C_VEL
LIN {X 0,Y 545.038,Z 326.214,A -85,B 0,C 180,E1 -3541.914,E2 -3541.914} C_VEL
LIN {X 0,Y 545.05,Z 326.216,A -85,B 0,C 180,E1 -3544.563,E2 -3544.563} C_VEL
LIN {X 0,Y 545.018,Z 326.219,A -85,B 0,C 180,E1 -3547.304,E2 -3547.304} C_VEL
LIN {X 0,Y 545.052,Z 326.212,A -85,B 0,C 180,E1 -3550.142,E2 -3550.142} C_VEL
LIN {X 0,Y 545.007,Z 326.222,A -85,B 0,C 180,E1 -3553.112,E2 -3553.112} C_VEL
LIN {X 0,Y 545.036,Z 326.214,A -85,B 0,C 180,E1 -3556.225,E2 -3556.225} C_VEL
LIN {X 0,Y 545.016,Z 326.224,A -85,B 0,C 180,E1 -3558.879,E2 -3558.879} C_VEL
LIN {X 0,Y 545.063,Z 326.217,A -85,B 0,C 180,E1 -3560.817,E2 -3560.817} C_VEL
LIN {X 0,Y 545.02,Z 326.215,A -85,B 0,C 180,E1 -3563.618,E2 -3563.618} C_VEL
LIN {X 0,Y 545.033,Z 326.215,A -85,B 0,C 180,E1 -3566.326,E2 -3566.326} C_VEL
LIN {X 0,Y 545.039,Z 326.219,A -85,B 0,C 180,E1 -3568.95,E2 -3568.95} C_VEL
LIN {X 0,Y 545.024,Z 326.214,A -85,B 0,C 180,E1 -3571.503,E2 -3571.503} C_VEL
LIN {X 0,Y 545.028,Z 326.209,A -85,B 0,C 180,E1 -3573.997,E2 -3573.997} C_VEL
LIN {X 0,Y 545.055,Z 326.215,A -85,B 0,C 180,E1 -3576.439,E2 -3576.439} C_VEL
LIN {X 0,Y 545.073,Z 326.205,A -85,B 0,C 180,E1 -3579.627,E2 -3579.627} C_VEL
LIN {X 0,Y 545.045,Z 326.219,A -85,B 0,C 180,E1 -3582.748,E2 -3582.748} C_VEL
LIN {X 0,Y 545.047,Z 326.211,A -85,B 0,C 180,E1 -3585.819,E2 -3585.819} C_VEL
LIN {X 0,Y 545.093,Z 326.212,A -85,B 0,C 180,E1 -3588.849,E2 -3588.849} C_VEL
LIN {X 0,Y 545.073,Z 326.208,A -85,B 0,C 180,E1 -3591.846,E2 -3591.846} C_VEL
LIN {X 0,Y 545.15,Z 326.203,A -85,B 0,C 180,E1 -3594.822,E2 -3594.822} C_VEL
LIN {X 0,Y 545.163,Z 326.197,A -85,B 0,C 180,E1 -3597.783,E2 -3597.783} C_VEL
LIN {X 0,Y 545.194,Z 326.2,A -85,B 0,C 180,E1 -3600.739,E2 -3600.739} C_VEL
LIN {X 0,Y 545.139,Z 326.202,A -85,B 0,C 180,E1 -3602.956,E2 -3602.956} C_VEL
LIN {X 0,Y 545.109,Z 326.205,A -85,B 0,C 180,E1 -3605.92,E2 -3605.92} C_VEL
LIN {X 0,Y 545.072,Z 326.211,A -85,B 0,C 180,E1 -3608.901,E2 -3608.901} C_VEL
LIN {X 0,Y 545.057,Z 326.212,A -85,B 0,C 180,E1 -3611.906,E2 -3611.906} C_VEL
LIN {X 0,Y 545.067,Z 326.211,A -85,B 0,C 180,E1 -3614.944,E2 -3614.944} C_VEL
LIN {X 0,Y 545.038,Z 326.215,A -85,B 0,C 180,E1 -3618.027,E2 -3618.027} C_VEL
LIN {X 0,Y 545.075,Z 326.216,A -85,B 0,C 180,E1 -3620.373,E2 -3620.373} C_VEL
LIN {X 0,Y 545.057,Z 326.207,A -85,B 0,C 180,E1 -3623.56,E2 -3623.56} C_VEL
LIN {X 0,Y 545.02,Z 326.219,A -85,B 0,C 180,E1 -3626.004,E2 -3626.004} C_VEL
LIN {X 0,Y 545.049,Z 326.212,A -85,B 0,C 180,E1 -3628.744,E2 -3628.744} C_VEL
LIN {X 0,Y 545.03,Z 326.215,A -85,B 0,C 180,E1 -3631.677,E2 -3631.677} C_VEL
LIN {X 0,Y 545.031,Z 326.219,A -85,B 0,C 180,E1 -3634.567,E2 -3634.567} C_VEL
LIN {X 0,Y 544.997,Z 326.218,A -85,B 0,C 180,E1 -3637.307,E2 -3637.307} C_VEL
LIN {X 0,Y 545.021,Z 326.222,A -85,B 0,C 180,E1 -3640.147,E2 -3640.147} C_VEL
LIN {X 0,Y 545.005,Z 326.217,A -85,B 0,C 180,E1 -3643.114,E2 -3643.114} C_VEL
LIN {X 0,Y 545.012,Z 326.225,A -85,B 0,C 180,E1 -3646.23,E2 -3646.23} C_VEL
LIN {X 0,Y 544.984,Z 326.221,A -85,B 0,C 180,E1 -3648.879,E2 -3648.879} C_VEL
LIN {X 0,Y 545.019,Z 326.22,A -85,B 0,C 180,E1 -3651.868,E2 -3651.868} C_VEL
LIN {X 0,Y 545.012,Z 326.221,A -85,B 0,C 180,E1 -3654.532,E2 -3654.532} C_VEL
LIN {X 0,Y 545.043,Z 326.213,A -85,B 0,C 180,E1 -3657.212,E2 -3657.212} C_VEL
LIN {X 0,Y 545.055,Z 326.215,A -85,B 0,C 180,E1 -3659.812,E2 -3659.812} C_VEL
LIN {X 0,Y 545.014,Z 326.218,A -85,B 0,C 180,E1 -3662.843,E2 -3662.843} C_VEL
LIN {X 0,Y 545.057,Z 326.281,A -85,B 0,C 180,E1 -3665.633,E2 -3665.633} C_VEL
LIN {X 0,Y 546.394,Z 333.022,A -85,B 0,C 180,E1 -3666.703,E2 -3666.703} C_VEL
LIN {X 0,Y 546.285,Z 345.157,A -85,B 0,C 180,E1 -3668.492,E2 -3668.492} C_VEL
LIN {X 0,Y 545.866,Z 364.022,A -85,B 0,C 180,E1 -3671.225,E2 -3671.225} C_VEL
LIN {X 0,Y 545.767,Z 371.943,A -85,B 0,C 180,E1 -3672.361,E2 -3672.361} C_VEL
LIN {X 0,Y 547.426,Z 381.387,A -85,B 0,C 180,E1 -3672.543,E2 -3672.543} C_VEL
LIN {X 0,Y 546.94,Z 508.701,A -85,B 0,C 180,E1 -3674.251,E2 -3674.251} C_VEL
LIN {X 0,Y 546.769,Z 523.046,A -85,B 0,C 180,E1 -3674.585,E2 -3674.585} C_VEL
LIN {X 0,Y 546.581,Z 536.699,A -85,B 0,C 180,E1 -3675.056,E2 -3675.056} C_VEL
LIN {X 0,Y 546.302,Z 549.895,A -85,B 0,C 180,E1 -3675.663,E2 -3675.663} C_VEL
LIN {X 0,Y 545.978,Z 562.694,A -85,B 0,C 180,E1 -3676.414,E2 -3676.414} C_VEL
LIN {X 0,Y 545.707,Z 574.322,A -85,B 0,C 180,E1 -3677.26,E2 -3677.26} C_VEL
LIN {X 0,Y 545.448,Z 585.131,A -85,B 0,C 180,E1 -3678.213,E2 -3678.213} C_VEL
LIN {X 0,Y 545.23,Z 594.717,A -85,B 0,C 180,E1 -3679.229,E2 -3679.229} C_VEL
LIN {X 0,Y 545.024,Z 603.565,A -85,B 0,C 180,E1 -3680.351,E2 -3680.351} C_VEL
LIN {X 0,Y 544.871,Z 612.042,A -85,B 0,C 180,E1 -3681.658,E2 -3681.658} C_VEL
LIN {X 0,Y 544.735,Z 618.868,A -85,B 0,C 180,E1 -3682.961,E2 -3682.961} C_VEL
LIN {X 0,Y 544.73,Z 623.572,A -85,B 0,C 180,E1 -3684.077,E2 -3684.077} C_VEL
LIN {X 0,Y 544.654,Z 628.45,A -85,B 0,C 180,E1 -3685.561,E2 -3685.561} C_VEL
LIN {X 0,Y 544.646,Z 631.838,A -85,B 0,C 180,E1 -3687.043,E2 -3687.043} C_VEL
LIN {X 0,Y 544.541,Z 633.837,A -85,B 0,C 180,E1 -3688.522,E2 -3688.522} C_VEL
LIN {X 0,Y 544.539,Z 634.5,A -85,B 0,C 180,E1 -3690.001,E2 -3690.001} C_VEL
LIN {X 0,Y 544.541,Z 633.833,A -85,B 0,C 180,E1 -3691.48,E2 -3691.48} C_VEL
LIN {X 0,Y 544.647,Z 631.83,A -85,B 0,C 180,E1 -3692.96,E2 -3692.96} C_VEL
LIN {X 0,Y 544.654,Z 628.441,A -85,B 0,C 180,E1 -3694.441,E2 -3694.441} C_VEL
LIN {X 0,Y 544.729,Z 623.565,A -85,B 0,C 180,E1 -3695.925,E2 -3695.925} C_VEL
LIN {X 0,Y 544.785,Z 617.049,A -85,B 0,C 180,E1 -3697.413,E2 -3697.413} C_VEL
LIN {X 0,Y 544.912,Z 609.796,A -85,B 0,C 180,E1 -3698.718,E2 -3698.718} C_VEL
LIN {X 0,Y 545.082,Z 600.814,A -85,B 0,C 180,E1 -3700.025,E2 -3700.025} C_VEL
LIN {X 0,Y 545.334,Z 591.383,A -85,B 0,C 180,E1 -3701.147,E2 -3701.147} C_VEL
LIN {X 0,Y 545.546,Z 580.942,A -85,B 0,C 180,E1 -3702.179,E2 -3702.179} C_VEL
LIN {X 0,Y 545.797,Z 569.413,A -85,B 0,C 180,E1 -3703.119,E2 -3703.119} C_VEL
LIN {X 0,Y 546.101,Z 556.618,A -85,B 0,C 180,E1 -3703.964,E2 -3703.964} C_VEL
LIN {X 0,Y 546.383,Z 544.13,A -85,B 0,C 180,E1 -3704.622,E2 -3704.622} C_VEL
LIN {X 0,Y 546.64,Z 531.741,A -85,B 0,C 180,E1 -3705.131,E2 -3705.131} C_VEL
LIN {X 0,Y 546.805,Z 517.692,A -85,B 0,C 180,E1 -3705.557,E2 -3705.557} C_VEL
LIN {X 0,Y 546.958,Z 504.048,A -85,B 0,C 180,E1 -3705.823,E2 -3705.823} C_VEL
LIN {X 0,Y 547.437,Z 381.105,A -85,B 0,C 180,E1 -3707.461,E2 -3707.461} C_VEL
LIN {X 0,Y 545.754,Z 371.875,A -85,B 0,C 180,E1 -3707.647,E2 -3707.647} C_VEL
LIN {X 0,Y 546.185,Z 350.533,A -85,B 0,C 180,E1 -3710.724,E2 -3710.724} C_VEL
LIN {X 0,Y 546.519,Z 334.357,A -85,B 0,C 180,E1 -3713.093,E2 -3713.093} C_VEL
LIN {X 0,Y 545.055,Z 326.217,A -85,B 0,C 180,E1 -3714.395,E2 -3714.395} C_VEL
LIN {X 0,Y 545.025,Z 326.22,A -85,B 0,C 180,E1 -3717.159,E2 -3717.159} C_VEL
LIN {X 0,Y 545.042,Z 326.215,A -85,B 0,C 180,E1 -3720.24,E2 -3720.24} C_VEL
LIN {X 0,Y 545.08,Z 326.213,A -85,B 0,C 180,E1 -3723.062,E2 -3723.062} C_VEL
LIN {X 0,Y 545.029,Z 326.218,A -85,B 0,C 180,E1 -3725.672,E2 -3725.672} C_VEL
LIN {X 0,Y 545.055,Z 326.211,A -85,B 0,C 180,E1 -3728.238,E2 -3728.238} C_VEL
LIN {X 0,Y 545.086,Z 326.209,A -85,B 0,C 180,E1 -3730.473,E2 -3730.473} C_VEL
LIN {X 0,Y 545.083,Z 326.214,A -85,B 0,C 180,E1 -3733.107,E2 -3733.107} C_VEL
LIN {X 0,Y 545.061,Z 326.213,A -85,B 0,C 180,E1 -3736.226,E2 -3736.226} C_VEL
LIN {X 0,Y 545.086,Z 326.213,A -85,B 0,C 180,E1 -3738.886,E2 -3738.886} C_VEL
LIN {X 0,Y 545.083,Z 326.213,A -85,B 0,C 180,E1 -3740.818,E2 -3740.818} C_VEL
LIN {X 0,Y 545.039,Z 326.213,A -85,B 0,C 180,E1 -3743.619,E2 -3743.619} C_VEL
LIN {X 0,Y 545.07,Z 326.217,A -85,B 0,C 180,E1 -3746.328,E2 -3746.328} C_VEL
LIN {X 0,Y 545.07,Z 326.211,A -85,B 0,C 180,E1 -3748.952,E2 -3748.952} C_VEL
LIN {X 0,Y 545.079,Z 326.213,A -85,B 0,C 180,E1 -3751.506,E2 -3751.506} C_VEL
LIN {X 0,Y 545.036,Z 326.217,A -85,B 0,C 180,E1 -3754.506,E2 -3754.506} C_VEL
LIN {X 0,Y 545.036,Z 326.22,A -85,B 0,C 180,E1 -3757.242,E2 -3757.242} C_VEL
LIN {X 0,Y 545.115,Z 326.412,A -85,B 0,C 180,E1 -3757.945,E2 -3757.945} C_VEL
LIN {X 0,Y 545.886,Z 332.212,A -85,B 0,C 180,E1 -3758.87,E2 -3758.87} C_VEL
LIN {X 0,Y 545.646,Z 349.217,A -85,B 0,C 180,E1 -3761.605,E2 -3761.605} C_VEL
LIN {X 0,Y 545.515,Z 360.166,A -85,B 0,C 180,E1 -3763.342,E2 -3763.342} C_VEL
LIN {X 0,Y 545.33,Z 373.17,A -85,B 0,C 180,E1 -3765.499,E2 -3765.499} C_VEL
LIN {X 0,Y 546.565,Z 381.724,A -85,B 0,C 180,E1 -3765.649,E2 -3765.649} C_VEL
LIN {X 0,Y 546.187,Z 480.249,A -85,B 0,C 180,E1 -3766.963,E2 -3766.963} C_VEL
LIN {X 0,Y 546.069,Z 493.725,A -85,B 0,C 180,E1 -3767.291,E2 -3767.291} C_VEL
LIN {X 0,Y 545.892,Z 505.89,A -85,B 0,C 180,E1 -3767.735,E2 -3767.735} C_VEL
LIN {X 0,Y 545.728,Z 518.133,A -85,B 0,C 180,E1 -3768.342,E2 -3768.342} C_VEL
LIN {X 0,Y 545.523,Z 529.059,A -85,B 0,C 180,E1 -3769.046,E2 -3769.046} C_VEL
LIN {X 0,Y 545.261,Z 539.549,A -85,B 0,C 180,E1 -3769.886,E2 -3769.886} C_VEL
LIN {X 0,Y 545.122,Z 548.182,A -85,B 0,C 180,E1 -3770.726,E2 -3770.726} C_VEL
LIN {X 0,Y 544.982,Z 556.064,A -85,B 0,C 180,E1 -3771.658,E2 -3771.658} C_VEL
LIN {X 0,Y 544.826,Z 563.854,A -85,B 0,C 180,E1 -3772.775,E2 -3772.775} C_VEL
LIN {X 0,Y 544.778,Z 570.943,A -85,B 0,C 180,E1 -3774.076,E2 -3774.076} C_VEL
LIN {X 0,Y 544.64,Z 575.711,A -85,B 0,C 180,E1 -3775.189,E2 -3775.189} C_VEL
LIN {X 0,Y 544.67,Z 579.302,A -85,B 0,C 180,E1 -3776.301,E2 -3776.301} C_VEL
LIN {X 0,Y 544.651,Z 581.163,A -85,B 0,C 180,E1 -3777.041,E2 -3777.041} C_VEL
LIN {X 0,Y 544.546,Z 583.636,A -85,B 0,C 180,E1 -3778.521,E2 -3778.521} C_VEL
LIN {X 0,Y 544.542,Z 584.273,A -85,B 0,C 180,E1 -3779.261,E2 -3779.261} C_VEL
LIN {X 0,Y 544.541,Z 584.496,A -85,B 0,C 180,E1 -3780,E2 -3780} C_VEL
LIN {X 0,Y 544.542,Z 584.306,A -85,B 0,C 180,E1 -3780.74,E2 -3780.74} C_VEL
LIN {X 0,Y 544.57,Z 582.739,A -85,B 0,C 180,E1 -3782.219,E2 -3782.219} C_VEL
LIN {X 0,Y 544.651,Z 581.359,A -85,B 0,C 180,E1 -3782.959,E2 -3782.959} C_VEL
LIN {X 0,Y 544.684,Z 578.513,A -85,B 0,C 180,E1 -3784.07,E2 -3784.07} C_VEL
LIN {X 0,Y 544.653,Z 574.609,A -85,B 0,C 180,E1 -3785.182,E2 -3785.182} C_VEL
LIN {X 0,Y 544.723,Z 569.366,A -85,B 0,C 180,E1 -3786.334,E2 -3786.334} C_VEL
LIN {X 0,Y 544.836,Z 563.232,A -85,B 0,C 180,E1 -3787.411,E2 -3787.411} C_VEL
LIN {X 0,Y 544.992,Z 555.335,A -85,B 0,C 180,E1 -3788.528,E2 -3788.528} C_VEL
LIN {X 0,Y 545.135,Z 547.233,A -85,B 0,C 180,E1 -3789.461,E2 -3789.461} C_VEL
LIN {X 0,Y 545.346,Z 537.42,A -85,B 0,C 180,E1 -3790.394,E2 -3790.394} C_VEL
LIN {X 0,Y 545.548,Z 527.647,A -85,B 0,C 180,E1 -3791.142,E2 -3791.142} C_VEL
LIN {X 0,Y 545.696,Z 516.885,A -85,B 0,C 180,E1 -3791.816,E2 -3791.816} C_VEL
LIN {X 0,Y 545.9,Z 504.651,A -85,B 0,C 180,E1 -3792.406,E2 -3792.406} C_VEL
LIN {X 0,Y 546.089,Z 492.01,A -85,B 0,C 180,E1 -3792.85,E2 -3792.85} C_VEL
LIN {X 0,Y 546.243,Z 478.797,A -85,B 0,C 180,E1 -3793.154,E2 -3793.154} C_VEL
LIN {X 0,Y 546.47,Z 380.126,A -85,B 0,C 180,E1 -3794.463,E2 -3794.463} C_VEL
LIN {X 0,Y 545.327,Z 373.072,A -85,B 0,C 180,E1 -3794.594,E2 -3794.594} C_VEL
LIN {X 0,Y 545.608,Z 353.885,A -85,B 0,C 180,E1 -3797.74,E2 -3797.74} C_VEL
LIN {X 0,Y 545.893,Z 335.527,A -85,B 0,C 180,E1 -3800.735,E2 -3800.735} C_VEL
LIN {X 0,Y 545.678,Z 329.41,A -85,B 0,C 180,E1 -3801.734,E2 -3801.734} C_VEL
LIN {X 0,Y 545.128,Z 327.816,A -85,B 0,C 180,E1 -3802.097,E2 -3802.097} C_VEL
LIN {X 0,Y 544.144,Z 326.97,A -85,B 0,C 180,E1 -3802.48,E2 -3802.48} C_VEL
LIN {X 0,Y 541.583,Z 326.646,A -85,B 0,C 180,E1 -3803.269,E2 -3803.269} C_VEL
LIN {X 0,Y 539.124,Z 326.958,A -85,B 0,C 180,E1 -3804.097,E2 -3804.097} C_VEL
LIN {X 0,Y 538.105,Z 327.083,A -85,B 0,C 180,E1 -3804.737,E2 -3804.737} C_VEL
LIN {X 0,Y 538.028,Z 327.088,A -85,B 0,C 180,E1 -3804.954,E2 -3804.954} C_VEL
LIN {X 0,Y 538.049,Z 327.084,A -85,B 0,C 180,E1 -3807.349,E2 -3807.349} C_VEL
LIN {X 0,Y 538.032,Z 327.089,A -85,B 0,C 180,E1 -3810.444,E2 -3810.444} C_VEL
LIN {X 0,Y 538.051,Z 327.084,A -85,B 0,C 180,E1 -3813.283,E2 -3813.283} C_VEL
LIN {X 0,Y 537.994,Z 327.098,A -85,B 0,C 180,E1 -3816.005,E2 -3816.005} C_VEL
LIN {X 0,Y 538.016,Z 327.088,A -85,B 0,C 180,E1 -3818.83,E2 -3818.83} C_VEL
LIN {X 0,Y 538.02,Z 327.096,A -85,B 0,C 180,E1 -3821.877,E2 -3821.877} C_VEL
LIN {X 0,Y 538.005,Z 327.089,A -85,B 0,C 180,E1 -3824.863,E2 -3824.863} C_VEL
LIN {X 0,Y 537.992,Z 327.094,A -85,B 0,C 180,E1 -3827.21,E2 -3827.21} C_VEL
LIN {X 0,Y 538.014,Z 327.088,A -85,B 0,C 180,E1 -3830.418,E2 -3830.418} C_VEL
LIN {X 0,Y 537.995,Z 327.094,A -85,B 0,C 180,E1 -3833.064,E2 -3833.064} C_VEL
LIN {X 0,Y 537.996,Z 327.094,A -85,B 0,C 180,E1 -3835.824,E2 -3835.824} C_VEL
LIN {X 0,Y 537.994,Z 327.092,A -85,B 0,C 180,E1 -3838.497,E2 -3838.497} C_VEL
LIN {X 0,Y 537.989,Z 327.099,A -85,B 0,C 180,E1 -3841.095,E2 -3841.095} C_VEL
LIN {X 0,Y 537.969,Z 327.1,A -85,B 0,C 180,E1 -3843.629,E2 -3843.629} C_VEL
LIN {X 0,Y 538.028,Z 327.142,A -85,B 0,C 180,E1 -3846.571,E2 -3846.571} C_VEL
LIN {X 0,Y 539.376,Z 334.423,A -85,B 0,C 180,E1 -3847.798,E2 -3847.798} C_VEL
LIN {X 0,Y 539.063,Z 349.636,A -85,B 0,C 180,E1 -3850.185,E2 -3850.185} C_VEL
LIN {X 0,Y 538.762,Z 362.442,A -85,B 0,C 180,E1 -3852.166,E2 -3852.166} C_VEL
LIN {X 0,Y 540.717,Z 373.661,A -85,B 0,C 180,E1 -3852.393,E2 -3852.393} C_VEL
LIN {X 0,Y 540.084,Z 498.512,A -85,B 0,C 180,E1 -3854.092,E2 -3854.092} C_VEL
LIN {X 0,Y 539.909,Z 510.97,A -85,B 0,C 180,E1 -3854.373,E2 -3854.373} C_VEL
LIN {X 0,Y 539.761,Z 524.843,A -85,B 0,C 180,E1 -3854.829,E2 -3854.829} C_VEL
LIN {X 0,Y 539.434,Z 539.013,A -85,B 0,C 180,E1 -3855.474,E2 -3855.474} C_VEL
LIN {X 0,Y 539.082,Z 550.489,A -85,B 0,C 180,E1 -3856.139,E2 -3856.139} C_VEL
LIN {X 0,Y 538.837,Z 560.049,A -85,B 0,C 180,E1 -3856.805,E2 -3856.805} C_VEL
LIN {X 0,Y 538.6,Z 569.317,A -85,B 0,C 180,E1 -3857.566,E2 -3857.566} C_VEL
LIN {X 0,Y 538.372,Z 578.106,A -85,B 0,C 180,E1 -3858.41,E2 -3858.41} C_VEL
LIN {X 0,Y 538.209,Z 585.846,A -85,B 0,C 180,E1 -3859.275,E2 -3859.275} C_VEL
LIN {X 0,Y 537.978,Z 593.162,A -85,B 0,C 180,E1 -3860.221,E2 -3860.221} C_VEL
LIN {X 0,Y 537.864,Z 599.449,A -85,B 0,C 180,E1 -3861.167,E2 -3861.167} C_VEL
LIN {X 0,Y 537.771,Z 604.862,A -85,B 0,C 180,E1 -3862.112,E2 -3862.112} C_VEL
LIN {X 0,Y 537.668,Z 610.295,A -85,B 0,C 180,E1 -3863.243,E2 -3863.243} C_VEL
LIN {X 0,Y 537.656,Z 614.741,A -85,B 0,C 180,E1 -3864.373,E2 -3864.373} C_VEL
LIN {X 0,Y 537.55,Z 618.291,A -85,B 0,C 180,E1 -3865.5,E2 -3865.5} C_VEL
LIN {X 0,Y 537.577,Z 620.213,A -85,B 0,C 180,E1 -3866.251,E2 -3866.251} C_VEL
LIN {X 0,Y 537.489,Z 622.934,A -85,B 0,C 180,E1 -3867.751,E2 -3867.751} C_VEL
LIN {X 0,Y 537.438,Z 624.244,A -85,B 0,C 180,E1 -3869.25,E2 -3869.25} C_VEL
LIN {X 0,Y 537.441,Z 624.496,A -85,B 0,C 180,E1 -3869.999,E2 -3869.999} C_VEL
LIN {X 0,Y 537.447,Z 623.841,A -85,B 0,C 180,E1 -3871.497,E2 -3871.497} C_VEL
LIN {X 0,Y 537.546,Z 621.851,A -85,B 0,C 180,E1 -3872.997,E2 -3872.997} C_VEL
LIN {X 0,Y 537.577,Z 620.436,A -85,B 0,C 180,E1 -3873.747,E2 -3873.747} C_VEL
LIN {X 0,Y 537.578,Z 616.304,A -85,B 0,C 180,E1 -3875.25,E2 -3875.25} C_VEL
LIN {X 0,Y 537.601,Z 612.616,A -85,B 0,C 180,E1 -3876.29,E2 -3876.29} C_VEL
LIN {X 0,Y 537.698,Z 607.226,A -85,B 0,C 180,E1 -3877.509,E2 -3877.509} C_VEL
LIN {X 0,Y 537.823,Z 601.131,A -85,B 0,C 180,E1 -3878.642,E2 -3878.642} C_VEL
LIN {X 0,Y 537.94,Z 595.14,A -85,B 0,C 180,E1 -3879.587,E2 -3879.587} C_VEL
LIN {X 0,Y 538.118,Z 588.155,A -85,B 0,C 180,E1 -3880.534,E2 -3880.534} C_VEL
LIN {X 0,Y 538.323,Z 580.426,A -85,B 0,C 180,E1 -3881.436,E2 -3881.436} C_VEL
LIN {X 0,Y 538.534,Z 571.386,A -85,B 0,C 180,E1 -3882.338,E2 -3882.338} C_VEL
LIN {X 0,Y 538.774,Z 562.47,A -85,B 0,C 180,E1 -3883.098,E2 -3883.098} C_VEL
LIN {X 0,Y 539.033,Z 553.347,A -85,B 0,C 180,E1 -3883.764,E2 -3883.764} C_VEL
LIN {X 0,Y 539.32,Z 542.434,A -85,B 0,C 180,E1 -3884.43,E2 -3884.43} C_VEL
LIN {X 0,Y 539.573,Z 530.957,A -85,B 0,C 180,E1 -3885.002,E2 -3885.002} C_VEL
LIN {X 0,Y 539.81,Z 519.987,A -85,B 0,C 180,E1 -3885.435,E2 -3885.435} C_VEL
LIN {X 0,Y 540.009,Z 507.897,A -85,B 0,C 180,E1 -3885.796,E2 -3885.796} C_VEL
LIN {X 0,Y 540.127,Z 494.072,A -85,B 0,C 180,E1 -3886.074,E2 -3886.074} C_VEL
LIN {X 0,Y 540.696,Z 373.022,A -85,B 0,C 180,E1 -3887.707,E2 -3887.707} C_VEL
LIN {X 0,Y 538.761,Z 362.336,A -85,B 0,C 180,E1 -3887.94,E2 -3887.94} C_VEL
LIN {X 0,Y 539.209,Z 342.627,A -85,B 0,C 180,E1 -3891.002,E2 -3891.002} C_VEL
LIN {X 0,Y 539.321,Z 334.4,A -85,B 0,C 180,E1 -3892.299,E2 -3892.299} C_VEL
LIN {X 0,Y 538.04,Z 327.092,A -85,B 0,C 180,E1 -3893.526,E2 -3893.526} C_VEL
LIN {X 0,Y 537.977,Z 327.096,A -85,B 0,C 180,E1 -3896.369,E2 -3896.369} C_VEL
LIN {X 0,Y 537.987,Z 327.101,A -85,B 0,C 180,E1 -3898.924,E2 -3898.924} C_VEL
LIN {X 0,Y 537.993,Z 327.092,A -85,B 0,C 180,E1 -3901.884,E2 -3901.884} C_VEL
LIN {X 0,Y 538,Z 327.095,A -85,B 0,C 180,E1 -3904.615,E2 -3904.615} C_VEL
LIN {X 0,Y 537.988,Z 327.097,A -85,B 0,C 180,E1 -3907.167,E2 -3907.167} C_VEL
LIN {X 0,Y 537.998,Z 327.09,A -85,B 0,C 180,E1 -3909.797,E2 -3909.797} C_VEL
LIN {X 0,Y 537.96,Z 327.102,A -85,B 0,C 180,E1 -3912.98,E2 -3912.98} C_VEL
LIN {X 0,Y 538.002,Z 327.089,A -85,B 0,C 180,E1 -3915.926,E2 -3915.926} C_VEL
LIN {X 0,Y 537.994,Z 327.094,A -85,B 0,C 180,E1 -3919.257,E2 -3919.257} C_VEL
LIN {X 0,Y 537.973,Z 327.091,A -85,B 0,C 180,E1 -3922.12,E2 -3922.12} C_VEL
LIN {X 0,Y 537.974,Z 327.1,A -85,B 0,C 180,E1 -3924.914,E2 -3924.914} C_VEL
LIN {X 0,Y 537.998,Z 327.086,A -85,B 0,C 180,E1 -3927.616,E2 -3927.616} C_VEL
LIN {X 0,Y 537.983,Z 327.093,A -85,B 0,C 180,E1 -3930.237,E2 -3930.237} C_VEL
LIN {X 0,Y 537.994,Z 327.093,A -85,B 0,C 180,E1 -3932.792,E2 -3932.792} C_VEL
LIN {X 0,Y 537.975,Z 327.094,A -85,B 0,C 180,E1 -3935.289,E2 -3935.289} C_VEL
LIN {X 0,Y 538,Z 327.09,A -85,B 0,C 180,E1 -3938.042,E2 -3938.042} C_VEL
LIN {X 0,Y 538.066,Z 327.079,A -85,B 0,C 180,E1 -3940.147,E2 -3940.147} C_VEL
LIN {X 0,Y 537.977,Z 327.093,A -85,B 0,C 180,E1 -3943.297,E2 -3943.297} C_VEL
LIN {X 0,Y 538.021,Z 327.086,A -85,B 0,C 180,E1 -3945.629,E2 -3945.629} C_VEL
LIN {X 0,Y 538.055,Z 327.091,A -85,B 0,C 180,E1 -3948.701,E2 -3948.701} C_VEL
LIN {X 0,Y 538.038,Z 327.083,A -85,B 0,C 180,E1 -3951.739,E2 -3951.739} C_VEL
LIN {X 0,Y 538.109,Z 327.081,A -85,B 0,C 180,E1 -3954.754,E2 -3954.754} C_VEL
LIN {X 0,Y 538.136,Z 327.073,A -85,B 0,C 180,E1 -3957.755,E2 -3957.755} C_VEL
LIN {X 0,Y 538.164,Z 327.075,A -85,B 0,C 180,E1 -3960.748,E2 -3960.748} C_VEL
LIN {X 0,Y 538.105,Z 327.078,A -85,B 0,C 180,E1 -3962.995,E2 -3962.995} C_VEL
LIN {X 0,Y 538.066,Z 327.083,A -85,B 0,C 180,E1 -3965.998,E2 -3965.998} C_VEL
LIN {X 0,Y 538.024,Z 327.088,A -85,B 0,C 180,E1 -3969.018,E2 -3969.018} C_VEL
LIN {X 0,Y 538.028,Z 327.089,A -85,B 0,C 180,E1 -3972.064,E2 -3972.064} C_VEL
LIN {X 0,Y 538.026,Z 327.087,A -85,B 0,C 180,E1 -3975.144,E2 -3975.144} C_VEL
LIN {X 0,Y 537.993,Z 327.096,A -85,B 0,C 180,E1 -3978.272,E2 -3978.272} C_VEL
LIN {X 0,Y 538.02,Z 327.089,A -85,B 0,C 180,E1 -3980.652,E2 -3980.652} C_VEL
LIN {X 0,Y 537.991,Z 327.09,A -85,B 0,C 180,E1 -3983.878,E2 -3983.878} C_VEL
LIN {X 0,Y 537.965,Z 327.102,A -85,B 0,C 180,E1 -3986.371,E2 -3986.371} C_VEL
LIN {X 0,Y 538.016,Z 327.085,A -85,B 0,C 180,E1 -3988.934,E2 -3988.934} C_VEL
LIN {X 0,Y 537.984,Z 327.094,A -85,B 0,C 180,E1 -3991.886,E2 -3991.886} C_VEL
LIN {X 0,Y 537.981,Z 327.097,A -85,B 0,C 180,E1 -3994.616,E2 -3994.616} C_VEL
LIN {X 0,Y 537.966,Z 327.097,A -85,B 0,C 180,E1 -3997.88,E2 -3997.88} C_VEL
LIN {X 0,Y 537.945,Z 327.098,A -85,B 0,C 180,E1 -4000.785,E2 -4000.785} C_VEL
LIN {X 0,Y 537.969,Z 327.096,A -85,B 0,C 180,E1 -4003.82,E2 -4003.82} C_VEL
LIN {X 0,Y 537.966,Z 327.102,A -85,B 0,C 180,E1 -4006.182,E2 -4006.182} C_VEL
LIN {X 0,Y 537.942,Z 327.097,A -85,B 0,C 180,E1 -4009.266,E2 -4009.266} C_VEL
LIN {X 0,Y 537.961,Z 327.104,A -85,B 0,C 180,E1 -4012.122,E2 -4012.122} C_VEL
LIN {X 0,Y 537.985,Z 327.093,A -85,B 0,C 180,E1 -4015.387,E2 -4015.387} C_VEL
LIN {X 0,Y 537.989,Z 327.099,A -85,B 0,C 180,E1 -4018.117,E2 -4018.117} C_VEL
LIN {X 0,Y 537.977,Z 327.092,A -85,B 0,C 180,E1 -4021.097,E2 -4021.097} C_VEL
LIN {X 0,Y 537.971,Z 327.098,A -85,B 0,C 180,E1 -4023.631,E2 -4023.631} C_VEL
LIN {X 0,Y 538.012,Z 327.164,A -85,B 0,C 180,E1 -4025.436,E2 -4025.436} C_VEL
LIN {X 0,Y 539.568,Z 335.661,A -85,B 0,C 180,E1 -4026.797,E2 -4026.797} C_VEL
LIN {X 0,Y 539.168,Z 355.015,A -85,B 0,C 180,E1 -4029.667,E2 -4029.667} C_VEL
LIN {X 0,Y 538.826,Z 371.801,A -85,B 0,C 180,E1 -4032.117,E2 -4032.117} C_VEL
LIN {X 0,Y 540.695,Z 383.258,A -85,B 0,C 180,E1 -4032.345,E2 -4032.345} C_VEL
LIN {X 0,Y 540.116,Z 508.634,A -85,B 0,C 180,E1 -4034.047,E2 -4034.047} C_VEL
LIN {X 0,Y 539.926,Z 523.145,A -85,B 0,C 180,E1 -4034.39,E2 -4034.39} C_VEL
LIN {X 0,Y 539.713,Z 535.858,A -85,B 0,C 180,E1 -4034.828,E2 -4034.828} C_VEL
LIN {X 0,Y 539.434,Z 548.069,A -85,B 0,C 180,E1 -4035.38,E2 -4035.38} C_VEL
LIN {X 0,Y 539.105,Z 561.231,A -85,B 0,C 180,E1 -4036.142,E2 -4036.142} C_VEL
LIN {X 0,Y 538.771,Z 573.125,A -85,B 0,C 180,E1 -4036.997,E2 -4036.997} C_VEL
LIN {X 0,Y 538.471,Z 583.991,A -85,B 0,C 180,E1 -4037.948,E2 -4037.948} C_VEL
LIN {X 0,Y 538.228,Z 594.717,A -85,B 0,C 180,E1 -4039.087,E2 -4039.087} C_VEL
LIN {X 0,Y 537.976,Z 603.564,A -85,B 0,C 180,E1 -4040.223,E2 -4040.223} C_VEL
LIN {X 0,Y 537.823,Z 612.042,A -85,B 0,C 180,E1 -4041.548,E2 -4041.548} C_VEL
LIN {X 0,Y 537.659,Z 618.868,A -85,B 0,C 180,E1 -4042.868,E2 -4042.868} C_VEL
LIN {X 0,Y 537.654,Z 624.963,A -85,B 0,C 180,E1 -4044.375,E2 -4044.375} C_VEL
LIN {X 0,Y 537.55,Z 628.45,A -85,B 0,C 180,E1 -4045.502,E2 -4045.502} C_VEL
LIN {X 0,Y 537.547,Z 631.838,A -85,B 0,C 180,E1 -4047.003,E2 -4047.003} C_VEL
LIN {X 0,Y 537.447,Z 633.837,A -85,B 0,C 180,E1 -4048.503,E2 -4048.503} C_VEL
LIN {X 0,Y 537.44,Z 634.5,A -85,B 0,C 180,E1 -4050.001,E2 -4050.001} C_VEL
LIN {X 0,Y 537.447,Z 633.834,A -85,B 0,C 180,E1 -4051.5,E2 -4051.5} C_VEL
LIN {X 0,Y 537.547,Z 631.83,A -85,B 0,C 180,E1 -4052.999,E2 -4052.999} C_VEL
LIN {X 0,Y 537.55,Z 628.44,A -85,B 0,C 180,E1 -4054.5,E2 -4054.5} C_VEL
LIN {X 0,Y 537.643,Z 623.565,A -85,B 0,C 180,E1 -4056.004,E2 -4056.004} C_VEL
LIN {X 0,Y 537.705,Z 617.049,A -85,B 0,C 180,E1 -4057.511,E2 -4057.511} C_VEL
LIN {X 0,Y 537.861,Z 609.796,A -85,B 0,C 180,E1 -4058.833,E2 -4058.833} C_VEL
LIN {X 0,Y 538.049,Z 600.814,A -85,B 0,C 180,E1 -4060.157,E2 -4060.157} C_VEL
LIN {X 0,Y 538.32,Z 591.382,A -85,B 0,C 180,E1 -4061.294,E2 -4061.294} C_VEL
LIN {X 0,Y 538.566,Z 580.929,A -85,B 0,C 180,E1 -4062.339,E2 -4062.339} C_VEL
LIN {X 0,Y 538.874,Z 569.384,A -85,B 0,C 180,E1 -4063.29,E2 -4063.29} C_VEL
LIN {X 0,Y 539.209,Z 556.575,A -85,B 0,C 180,E1 -4064.147,E2 -4064.147} C_VEL
LIN {X 0,Y 539.512,Z 544.075,A -85,B 0,C 180,E1 -4064.813,E2 -4064.813} C_VEL
LIN {X 0,Y 539.789,Z 530.842,A -85,B 0,C 180,E1 -4065.359,E2 -4065.359} C_VEL
LIN {X 0,Y 540.017,Z 516.696,A -85,B 0,C 180,E1 -4065.782,E2 -4065.782} C_VEL
LIN {X 0,Y 540.146,Z 502.456,A -85,B 0,C 180,E1 -4066.052,E2 -4066.052} C_VEL
LIN {X 0,Y 540.668,Z 382.704,A -85,B 0,C 180,E1 -4067.664,E2 -4067.664} C_VEL
LIN {X 0,Y 538.794,Z 371.805,A -85,B 0,C 180,E1 -4067.884,E2 -4067.884} C_VEL
LIN {X 0,Y 539.269,Z 350.471,A -85,B 0,C 180,E1 -4071.002,E2 -4071.002} C_VEL
LIN {X 0,Y 539.599,Z 335.645,A -85,B 0,C 180,E1 -4073.204,E2 -4073.204} C_VEL
LIN {X 0,Y 538.016,Z 327.094,A -85,B 0,C 180,E1 -4074.614,E2 -4074.614} C_VEL
LIN {X 0,Y 537.992,Z 327.098,A -85,B 0,C 180,E1 -4077.338,E2 -4077.338} C_VEL
LIN {X 0,Y 538.007,Z 327.091,A -85,B 0,C 180,E1 -4080.44,E2 -4080.44} C_VEL
LIN {X 0,Y 538.051,Z 327.091,A -85,B 0,C 180,E1 -4083.283,E2 -4083.283} C_VEL
LIN {X 0,Y 537.994,Z 327.091,A -85,B 0,C 180,E1 -4086.006,E2 -4086.006} C_VEL
LIN {X 0,Y 538.018,Z 327.092,A -85,B 0,C 180,E1 -4088.831,E2 -4088.831} C_VEL
LIN {X 0,Y 538.035,Z 327.086,A -85,B 0,C 180,E1 -4091.774,E2 -4091.774} C_VEL
LIN {X 0,Y 538.034,Z 327.094,A -85,B 0,C 180,E1 -4094.86,E2 -4094.86} C_VEL
LIN {X 0,Y 538.033,Z 327.088,A -85,B 0,C 180,E1 -4098.122,E2 -4098.122} C_VEL
LIN {X 0,Y 538.037,Z 327.092,A -85,B 0,C 180,E1 -4100.416,E2 -4100.416} C_VEL
LIN {X 0,Y 538.023,Z 327.089,A -85,B 0,C 180,E1 -4103.067,E2 -4103.067} C_VEL
LIN {X 0,Y 538.022,Z 327.09,A -85,B 0,C 180,E1 -4105.827,E2 -4105.827} C_VEL
LIN {X 0,Y 538.013,Z 327.095,A -85,B 0,C 180,E1 -4108.499,E2 -4108.499} C_VEL
LIN {X 0,Y 538.023,Z 327.091,A -85,B 0,C 180,E1 -4111.098,E2 -4111.098} C_VEL
LIN {X 0,Y 537.986,Z 327.1,A -85,B 0,C 180,E1 -4113.63,E2 -4113.63} C_VEL
LIN {X 0,Y 538.011,Z 327.097,A -85,B 0,C 180,E1 -4116.123,E2 -4116.123} C_VEL
LIN {X 0,Y 538.059,Z 327.236,A -85,B 0,C 180,E1 -4117.849,E2 -4117.849} C_VEL
LIN {X 0,Y 538.893,Z 333.179,A -85,B 0,C 180,E1 -4118.783,E2 -4118.783} C_VEL
LIN {X 0,Y 538.697,Z 349.201,A -85,B 0,C 180,E1 -4121.359,E2 -4121.359} C_VEL
LIN {X 0,Y 538.549,Z 361.538,A -85,B 0,C 180,E1 -4123.316,E2 -4123.316} C_VEL
LIN {X 0,Y 538.333,Z 373.42,A -85,B 0,C 180,E1 -4125.311,E2 -4125.311} C_VEL
LIN {X 0,Y 539.673,Z 381.946,A -85,B 0,C 180,E1 -4125.471,E2 -4125.471} C_VEL
LIN {X 0,Y 539.256,Z 480.62,A -85,B 0,C 180,E1 -4126.816,E2 -4126.816} C_VEL
LIN {X 0,Y 539.127,Z 494.095,A -85,B 0,C 180,E1 -4127.149,E2 -4127.149} C_VEL
LIN {X 0,Y 538.932,Z 506.822,A -85,B 0,C 180,E1 -4127.622,E2 -4127.622} C_VEL
LIN {X 0,Y 538.755,Z 518.926,A -85,B 0,C 180,E1 -4128.238,E2 -4128.238} C_VEL
LIN {X 0,Y 538.517,Z 530.433,A -85,B 0,C 180,E1 -4128.997,E2 -4128.997} C_VEL
LIN {X 0,Y 538.23,Z 540.651,A -85,B 0,C 180,E1 -4129.847,E2 -4129.847} C_VEL
LIN {X 0,Y 538.083,Z 549.965,A -85,B 0,C 180,E1 -4130.793,E2 -4130.793} C_VEL
LIN {X 0,Y 537.886,Z 557.517,A -85,B 0,C 180,E1 -4131.737,E2 -4131.737} C_VEL
LIN {X 0,Y 537.745,Z 564.982,A -85,B 0,C 180,E1 -4132.868,E2 -4132.868} C_VEL
LIN {X 0,Y 537.696,Z 570.941,A -85,B 0,C 180,E1 -4133.998,E2 -4133.998} C_VEL
LIN {X 0,Y 537.55,Z 575.708,A -85,B 0,C 180,E1 -4135.125,E2 -4135.125} C_VEL
LIN {X 0,Y 537.592,Z 579.3,A -85,B 0,C 180,E1 -4136.252,E2 -4136.252} C_VEL
LIN {X 0,Y 537.552,Z 581.159,A -85,B 0,C 180,E1 -4137.002,E2 -4137.002} C_VEL
LIN {X 0,Y 537.489,Z 582.596,A -85,B 0,C 180,E1 -4137.752,E2 -4137.752} C_VEL
LIN {X 0,Y 537.442,Z 584.272,A -85,B 0,C 180,E1 -4139.251,E2 -4139.251} C_VEL
LIN {X 0,Y 537.442,Z 584.496,A -85,B 0,C 180,E1 -4140,E2 -4140} C_VEL
LIN {X 0,Y 537.442,Z 584.301,A -85,B 0,C 180,E1 -4140.749,E2 -4140.749} C_VEL
LIN {X 0,Y 537.489,Z 582.734,A -85,B 0,C 180,E1 -4142.248,E2 -4142.248} C_VEL
LIN {X 0,Y 537.552,Z 581.352,A -85,B 0,C 180,E1 -4142.998,E2 -4142.998} C_VEL
LIN {X 0,Y 537.604,Z 578.508,A -85,B 0,C 180,E1 -4144.123,E2 -4144.123} C_VEL
LIN {X 0,Y 537.587,Z 574.601,A -85,B 0,C 180,E1 -4145.251,E2 -4145.251} C_VEL
LIN {X 0,Y 537.68,Z 568.532,A -85,B 0,C 180,E1 -4146.586,E2 -4146.586} C_VEL
LIN {X 0,Y 537.809,Z 562.022,A -85,B 0,C 180,E1 -4147.698,E2 -4147.698} C_VEL
LIN {X 0,Y 537.959,Z 553.895,A -85,B 0,C 180,E1 -4148.83,E2 -4148.83} C_VEL
LIN {X 0,Y 538.133,Z 545.465,A -85,B 0,C 180,E1 -4149.775,E2 -4149.775} C_VEL
LIN {X 0,Y 538.369,Z 535.149,A -85,B 0,C 180,E1 -4150.721,E2 -4150.721} C_VEL
LIN {X 0,Y 538.621,Z 524.175,A -85,B 0,C 180,E1 -4151.53,E2 -4151.53} C_VEL
LIN {X 0,Y 538.839,Z 511.78,A -85,B 0,C 180,E1 -4152.237,E2 -4152.237} C_VEL
LIN {X 0,Y 539.055,Z 499.622,A -85,B 0,C 180,E1 -4152.758,E2 -4152.758} C_VEL
LIN {X 0,Y 539.231,Z 486.207,A -85,B 0,C 180,E1 -4153.16,E2 -4153.16} C_VEL
LIN {X 0,Y 539.331,Z 473.112,A -85,B 0,C 180,E1 -4153.398,E2 -4153.398} C_VEL
LIN {X 0,Y 539.566,Z 380.799,A -85,B 0,C 180,E1 -4154.639,E2 -4154.639} C_VEL
LIN {X 0,Y 538.343,Z 373.239,A -85,B 0,C 180,E1 -4154.798,E2 -4154.798} C_VEL
LIN {X 0,Y 538.643,Z 354.244,A -85,B 0,C 180,E1 -4157.922,E2 -4157.922} C_VEL
LIN {X 0,Y 538.918,Z 335.365,A -85,B 0,C 180,E1 -4161.016,E2 -4161.016} C_VEL
LIN {X 0,Y 538.755,Z 330.927,A -85,B 0,C 180,E1 -4161.749,E2 -4161.749} C_VEL
LIN {X 0,Y 538.026,Z 327.095,A -85,B 0,C 180,E1 -4162.412,E2 -4162.412} C_VEL
LIN {X 0,Y 538.028,Z 327.088,A -85,B 0,C 180,E1 -4164.954,E2 -4164.954} C_VEL
LIN {X 0,Y 537.376,Z 327.17,A -85,B 0,C 180,E1 -4165.578,E2 -4165.578} C_VEL
LIN {X 0,Y 534.519,Z 327.528,A -85,B 0,C 180,E1 -4166.592,E2 -4166.592} C_VEL
